// TIA Portal project "OPCUA@SUP_HandsOnProject_V16_Referent" (V16)

(* hardware
DEVICE "S71500/ET200MP-Station_1"  S7-1500 station
   slot 0: "Profilschiene_0"  Rack  6ES7 590-1***0-0AA0
   slot 1: "OPCServer@SUP"  CPU 1518-4 PN/DP  6ES7 518-4AP00-0AB0  V2.8
      slot 3: "CPU-Display_1"  6ES7591-1BA00-0AA0
      slot 32768: "PROFINET-Schnittstelle_1"  X1
      slot 33024: "PROFINET-Schnittstelle_2"  X2
      slot 33280: "PROFINET-Schnittstelle GBIT_3"  X3
      slot 34817: "Virtual CP interface port_1"  Virtual CP interface port  Virtual CP interface port
DEVICE "S71500/ET200MP-Station_2"  S7-1500 station
   slot 0: "Profilschiene_0"  Rack  6ES7 590-1***0-0AA0
   slot 1: "ZOPCClient@SUP"  CPU 1518-4 PN/DP  6ES7 518-4AP00-0AB0  V2.8
      slot 3: "CPU-Display_1"  6ES7591-1BA00-0AA0
      slot 32768: "PROFINET-Schnittstelle_1"  X1
      slot 33024: "PROFINET-Schnittstelle_2"  X2
      slot 33280: "PROFINET-Schnittstelle GBIT_3"  X3
      slot 34817: "Virtual CP interface port_1"  Virtual CP interface port  Virtual CP interface port
*)

// ===== PLC "OPCServer@SUP"  CPU 1518-4 PN/DP =====

VAR_GLOBAL   // PLC tag table "StandardVariablentabelle"
   "ClockByte" AT %MB0 : Byte;
   "Clock10Hz" AT %M0.0 : Bool;
   "Clock5Hz" AT %M0.1 : Bool;
   "Clock2.5Hz" AT %M0.2 : Bool;
   "Clock2Hz" AT %M0.3 : Bool;
   "Clock1.25Hz" AT %M0.4 : Bool;
   "Clock1Hz" AT %M0.5 : Bool;
   "Clock0.625Hz" AT %M0.6 : Bool;
   "Clock0.5Hz" AT %M0.7 : Bool;
   "SystemByte" AT %MB1 : Byte;
   "FirstScan" AT %M1.0 : Bool;
   "DiagStatusUpdate" AT %M1.1 : Bool;
   "AlwaysTRUE" AT %M1.2 : Bool;
   "AlwaysFALSE" AT %M1.3 : Bool;
END_VAR

VAR_GLOBAL   // PLC tag table "AnalogTags"
   "AI0" AT %EW4 : Word;
   "AI1" AT %EW9 : Word;
   "AI2" AT %EW11 : Word;
   "AI3" AT %EW13 : Word;
   "AI4" AT %EW15 : Word;
   "AI5" AT %EW14 : Word;
   "AI6" AT %EW16 : Word;
   "AI7" AT %EW18 : Word;
   "AO0" AT %AW4 : Word;
   "AO1" AT %AW6 : Word;
   "AO2" AT %AW8 : Word;
   "AO3" AT %AW10 : Word;
END_VAR

VAR_GLOBAL   // PLC tag table "CounterTags"
   "Z1" AT %Z1 : Counter;
   "Z2" AT %Z2 : Counter;
   "Z3" AT %Z3 : Counter;
   "Z4" AT %Z4 : Counter;
   "Z5" AT %Z5 : Counter;
   "Z7" AT %Z7 : Counter;
   "Z8" AT %Z8 : Counter;
   "Z9" AT %Z9 : Counter;
   "Z10" AT %Z10 : Counter;
   "ZTest" AT %Z100 : Counter;
   "Z6" AT %Z6 : Counter;
   "Z500" AT %Z500 : Counter;
   "Z1000" AT %Z1000 : Counter;
   "Z1023" AT %Z1023 : Counter;
   "Z1024" AT %Z1024 : Counter;
   "Z2047" AT %Z2047 : Counter;
END_VAR

VAR_GLOBAL   // PLC tag table "DigitalInputTags"
   "DI01" AT %E0.1 : Bool;
   "DI02" AT %E0.2 : Bool;
   "DI03" AT %E0.3 : Bool;
   "DI04" AT %E0.4 : Bool;
   "DI05" AT %E0.5 : Bool;
   "DI06" AT %E0.6 : Bool;
   "DI07" AT %E0.7 : Bool;
   "DI11" AT %E1.1 : Bool;
   "DI12" AT %E1.2 : Bool;
   "DI13" AT %E1.3 : Bool;
   "DI14" AT %E1.4 : Bool;
   "DI15" AT %E1.5 : Bool;
   "DI16" AT %E1.6 : Bool;
   "DI17" AT %E1.7 : Bool;
   "DI20" AT %E2.0 : Bool;
   "DI21" AT %E2.1 : Bool;
   "DI22" AT %E2.2 : Bool;
   "DI23" AT %E2.3 : Bool;
   "DI24" AT %E2.4 : Bool;
   "DI25" AT %E2.5 : Bool;
   "DI26" AT %E2.6 : Bool;
   "DI27" AT %E2.7 : Bool;
   "DI30" AT %E3.0 : Bool;
   "DI31" AT %E3.1 : Bool;
   "DI32" AT %E3.2 : Bool;
   "DI33" AT %E3.3 : Bool;
   "DI34" AT %E3.4 : Bool;
   "DI35" AT %E3.5 : Bool;
   "DI36" AT %E3.6 : Bool;
   "DI37" AT %E3.7 : Bool;
   "DI10" AT %E1.0 : Bool;
   "DI00" AT %E0.0 : Bool;
   "DI1" AT %EB1 : Byte;
   "DI300" AT %EB300 : Byte;
   "DI310W" AT %EW310 : Word;
   "DI320D" AT %ED320 : DWord;
   "DI3300" AT %E330.0 : Bool;
   "DI340L" AT %E340.0 : LWord;
   "DI0" AT %EB0 : Byte;
END_VAR

VAR_GLOBAL   // PLC tag table "DigitalOutputTags"
   "DO01" AT %A0.1 : Bool;
   "DO02" AT %A0.2 : Bool;
   "DO04" AT %A0.4 : Bool;
   "DO05" AT %A0.5 : Bool;
   "DO06" AT %A0.6 : Bool;
   "DO07" AT %A0.7 : Bool;
   "DO10" AT %A1.0 : Bool;
   "DO11" AT %A1.1 : Bool;
   "DO12" AT %A1.2 : Bool;
   "DO13" AT %A1.3 : Bool;
   "DO14" AT %A1.4 : Bool;
   "DO15" AT %A1.5 : Bool;
   "DO16" AT %A1.6 : Bool;
   "DO17" AT %A1.7 : Bool;
   "DO20" AT %A2.0 : Bool;
   "DO21" AT %A2.1 : Bool;
   "DO22" AT %A2.2 : Bool;
   "DO23" AT %A2.3 : Bool;
   "DO24" AT %A2.4 : Bool;
   "DO25" AT %A2.5 : Bool;
   "DO26" AT %A2.6 : Bool;
   "DO27" AT %A2.7 : Bool;
   "DO30" AT %A3.0 : Bool;
   "DO31" AT %A3.1 : Bool;
   "DO32" AT %A3.2 : Bool;
   "DO33" AT %A3.3 : Bool;
   "DO34" AT %A3.4 : Bool;
   "DO35" AT %A3.5 : Bool;
   "DO36" AT %A3.6 : Bool;
   "DO37" AT %A3.7 : Bool;
   "DO300" AT %AB300 : Byte;
   "DO00" AT %A0.0 : Bool;
   "DO03" AT %A0.3 : Bool;
   "DO120" AT %A12.0 : Bool;
   "DO1" AT %AB1 : Byte;
   "DO0" AT %AB0 : Byte;
   "DOW0" AT %AW0 : Word;
   "DOW2" AT %AW2 : Word;
   "DO310W" AT %AW310 : Word;
   "DO320D" AT %AD320 : DWord;
   "DO3300" AT %A330.0 : Bool;
   "DO340L" AT %A340.0 : LWord;
END_VAR

VAR_GLOBAL   // PLC tag table "MerkerTags"
   "M1000" AT %M100.0 : Bool;
   "M1001" AT %M100.1 : Bool;
   "M1002" AT %M100.2 : Bool;
   "M1003" AT %M100.3 : Bool;
   "M1004" AT %M100.4 : Bool;
   "M1005" AT %M100.5 : Bool;
   "M1006" AT %M100.6 : Bool;
   "M1007" AT %M100.7 : Bool;
   "MB110" AT %MB110 : Byte;
   "MW120" AT %MW120 : Word;
   "MD130" AT %MD130 : DWord;
   "CharMb" AT %MB200 : Char;
   "DateMw" AT %MW202 : Date;
   "DintMd" AT %MD204 : DInt;
   "IntMw" AT %MW208 : Int;
   "LdtMl" AT %M210.0 : LDT;
   "LintMl" AT %M218.0 : LInt;
   "LrealMl" AT %M226.0 : LReal;
   "LtimeMl" AT %M234.0 : LTime;
   "LtodMl" AT %M242.0 : LTime_Of_Day;
   "LwordMl" AT %M250.0 : LWord;
   "RealMd" AT %MD258 : Real;
   "S5timeMw" AT %MW262 : S5Time;
   "SintMb" AT %MB264 : SInt;
   "TimeMd" AT %MD266 : Time;
   "TodMd" AT %MD270 : Time_Of_Day;
   "UdintMd" AT %MD274 : UDInt;
   "UintMw" AT %MW278 : UInt;
   "UlintMl" AT %M280.0 : ULInt;
   "UsintMb" AT %MB288 : USInt;
   "Z1MB" AT %MB500 : Byte;
   "Z2MB" AT %MB501 : Byte;
   "ZTestMx" AT %M502.0 : Bool;
   "Z6FP" AT %M502.1 : Bool;
   "Z7FP" AT %M502.2 : Bool;
   "Z8FP" AT %M502.3 : Bool;
   "Z9FP" AT %M502.4 : Bool;
   "Z10FP" AT %M502.5 : Bool;
   "TremMx" AT %M105.0 : Bool;
   "IintMw400" AT %MW400 : Int;
END_VAR

VAR_GLOBAL   // PLC tag table "TimerTags"
   "T1" AT %T1 : Timer;
   "T3" AT %T3 : Timer;
   "T4" AT %T4 : Timer;
   "T5" AT %T5 : Timer;
   "T6" AT %T6 : Timer;
   "T7" AT %T7 : Timer;
   "T9" AT %T9 : Timer;
   "T10" AT %T10 : Timer;
   "T2" AT %T2 : Timer;
   "T8" AT %T8 : Timer;
   "T20" AT %T20 : Timer;
   "T40" AT %T40 : Timer;
   "T60" AT %T60 : Timer;
   "T80" AT %T80 : Timer;
   "T100" AT %T100 : Timer;
   "T200" AT %T200 : Timer;
   "T500" AT %T500 : Timer;
   "T1000" AT %T1000 : Timer;
   "T2000" AT %T2000 : Timer;
   "T99" AT %T99 : Timer;
   "T85" AT %T85 : Timer;
   "T86" AT %T86 : Timer;
   "T2047" AT %T2047 : Timer;
END_VAR

VAR_GLOBAL CONSTANT   // PLC tag table "Tag table from XML_1"
   "OpcUa_Good" : DWord := 16#00000000;   // Everything is as expected.
   "OpcUa_Uncertain" : DWord := 16#40000000;   // Something unexpected occurred but the results still maybe useable.
   "OpcUa_Bad" : DWord := 16#80000000;   // An error occurred.
   "OpcUa_BadUnexpectedError" : DWord := 16#80010000;   // An unexpected error occurred.
   "OpcUa_BadInternalError" : DWord := 16#80020000;   // An internal error occurred as a result of a programming or configuration error.
   "OpcUa_BadOutOfMemory" : DWord := 16#80030000;   // Not enough memory to complete the operation.
   "OpcUa_BadResourceUnavailable" : DWord := 16#80040000;   // An operating system resource is not available.
   "OpcUa_BadCommunicationError" : DWord := 16#80050000;   // A low level communication error occurred.
   "OpcUa_BadEncodingError" : DWord := 16#80060000;   // Encoding halted because of invalid data in the objects being serialized.
   "OpcUa_BadDecodingError" : DWord := 16#80070000;   // Decoding halted because of invalid data in the stream.
   "OpcUa_BadEncodingLimitsExceeded" : DWord := 16#80080000;   // The message encoding/decoding limits imposed by the stack have been exceeded.
   "OpcUa_BadRequestTooLarge" : DWord := 16#80B80000;   // The request message size exceeds limits set by the server.
   "OpcUa_BadResponseTooLarge" : DWord := 16#80B90000;   // The response message size exceeds limits set by the client.
   "OpcUa_BadUnknownResponse" : DWord := 16#80090000;   // An unrecognized response was received from the server.
   "OpcUa_BadTimeout" : DWord := 16#800A0000;   // The operation timed out.
   "OpcUa_BadServiceUnsupported" : DWord := 16#800B0000;   // The server does not support the requested service.
   "OpcUa_BadShutdown" : DWord := 16#800C0000;   // The operation was cancelled because the application is shutting down.
   "OpcUa_BadServerNotConnected" : DWord := 16#800D0000;   // The operation could not complete because the client is not connected to the server.
   "OpcUa_BadServerHalted" : DWord := 16#800E0000;   // The server has stopped and cannot process any requests.
   "OpcUa_BadNothingToDo" : DWord := 16#800F0000;   // There was nothing to do because the client passed a list of operations with no elements.
   "OpcUa_BadTooManyOperations" : DWord := 16#80100000;   // The request could not be processed because it specified too many operations.
   "OpcUa_BadTooManyMonitoredItems" : DWord := 16#80DB0000;   // The request could not be processed because there are too many monitored items in the subscription.
   "OpcUa_BadDataTypeIdUnknown" : DWord := 16#80110000;   // The extension object cannot be (de)serialized because the data type id is not recognized.
   "OpcUa_BadCertificateInvalid" : DWord := 16#80120000;   // The certificate provided as a parameter is not valid.
   "OpcUa_BadSecurityChecksFailed" : DWord := 16#80130000;   // An error occurred verifying security.
   "OpcUa_BadCertificateTimeInvalid" : DWord := 16#80140000;   // The certificate has expired or is not yet valid.
   "OpcUa_BadCertificateIssuerTimeInvalid" : DWord := 16#80150000;   // An issuer certificate has expired or is not yet valid.
   "OpcUa_BadCertificateHostNameInvalid" : DWord := 16#80160000;   // The HostName used to connect to a server does not match a HostName in the certificate.
   "OpcUa_BadCertificateUriInvalid" : DWord := 16#80170000;   // The URI specified in the ApplicationDescription does not match the URI in the certificate.
   "OpcUa_BadCertificateUseNotAllowed" : DWord := 16#80180000;   // The certificate may not be used for the requested operation.
   "OpcUa_BadCertificateIssuerUseNotAllowed" : DWord := 16#80190000;   // The issuer certificate may not be used for the requested operation.
   "OpcUa_BadCertificateUntrusted" : DWord := 16#801A0000;   // The certificate is not trusted.
   "OpcUa_BadCertificateRevocationUnknown" : DWord := 16#801B0000;   // It was not possible to determine if the certificate has been revoked.
   "OpcUa_BadCertificateIssuerRevocationUnknown" : DWord := 16#801C0000;   // It was not possible to determine if the issuer certificate has been revoked.
   "OpcUa_BadCertificateRevoked" : DWord := 16#801D0000;   // The certificate has been revoked.
   "OpcUa_BadCertificateIssuerRevoked" : DWord := 16#801E0000;   // The issuer certificate has been revoked.
   "OpcUa_BadCertificateChainIncomplete" : DWord := 16#810D0000;   // The certificate chain is incomplete.
   "OpcUa_BadUserAccessDenied" : DWord := 16#801F0000;   // User does not have permission to perform the requested operation.
   "OpcUa_BadIdentityTokenInvalid" : DWord := 16#80200000;   // The user identity token is not valid.
   "OpcUa_BadIdentityTokenRejected" : DWord := 16#80210000;   // The user identity token is valid but the server has rejected it.
   "OpcUa_BadSecureChannelIdInvalid" : DWord := 16#80220000;   // The specified secure channel is no longer valid.
   "OpcUa_BadInvalidTimestamp" : DWord := 16#80230000;   // The timestamp is outside the range allowed by the server.
   "OpcUa_BadNonceInvalid" : DWord := 16#80240000;   // The nonce does appear to be not a random value or it is not the correct length.
   "OpcUa_BadSessionIdInvalid" : DWord := 16#80250000;   // The session id is not valid.
   "OpcUa_BadSessionClosed" : DWord := 16#80260000;   // The session was closed by the client.
   "OpcUa_BadSessionNotActivated" : DWord := 16#80270000;   // The session cannot be used because ActivateSession has not been called.
   "OpcUa_BadSubscriptionIdInvalid" : DWord := 16#80280000;   // The subscription id is not valid.
   "OpcUa_BadRequestHeaderInvalid" : DWord := 16#802A0000;   // The header for the request is missing or invalid.
   "OpcUa_BadTimestampsToReturnInvalid" : DWord := 16#802B0000;   // The timestamps to return parameter is invalid.
   "OpcUa_BadRequestCancelledByClient" : DWord := 16#802C0000;   // The request was cancelled by the client.
   "OpcUa_BadTooManyArguments" : DWord := 16#80E50000;   // Too many arguments were provided.
   "OpcUa_BadLicenseExpired" : DWord := 16#810E0000;   // The server requires a license to operate in general or to perform a service or operation, but existing license is expired.
   "OpcUa_BadLicenseLimitsExceeded" : DWord := 16#810F0000;   // The server has limits on number of allowed operations / objects, based on installed licenses, and these limits where exceeded.
   "OpcUa_BadLicenseNotAvailable" : DWord := 16#81100000;   // The server does not have a license which is required to operate in general or to perform a service or operation.
   "OpcUa_GoodSubscriptionTransferred" : DWord := 16#002D0000;   // The subscription was transferred to another session.
   "OpcUa_GoodCompletesAsynchronously" : DWord := 16#002E0000;   // The processing will complete asynchronously.
   "OpcUa_GoodOverload" : DWord := 16#002F0000;   // Sampling has slowed down due to resource limitations.
   "OpcUa_GoodClamped" : DWord := 16#00300000;   // The value written was accepted but was clamped.
   "OpcUa_BadNoCommunication" : DWord := 16#80310000;   // Communication with the data source is defined, but not established, and there is no last known value available.
   "OpcUa_BadWaitingForInitialData" : DWord := 16#80320000;   // Waiting for the server to obtain values from the underlying data source.
   "OpcUa_BadNodeIdInvalid" : DWord := 16#80330000;   // The syntax of the node id is not valid.
   "OpcUa_BadNodeIdUnknown" : DWord := 16#80340000;   // The node id refers to a node that does not exist in the server address space.
   "OpcUa_BadAttributeIdInvalid" : DWord := 16#80350000;   // The attribute is not supported for the specified Node.
   "OpcUa_BadIndexRangeInvalid" : DWord := 16#80360000;   // The syntax of the index range parameter is invalid.
   "OpcUa_BadIndexRangeNoData" : DWord := 16#80370000;   // No data exists within the range of indexes specified.
   "OpcUa_BadDataEncodingInvalid" : DWord := 16#80380000;   // The data encoding is invalid.
   "OpcUa_BadDataEncodingUnsupported" : DWord := 16#80390000;   // The server does not support the requested data encoding for the node.
   "OpcUa_BadNotReadable" : DWord := 16#803A0000;   // The access level does not allow reading or subscribing to the Node.
   "OpcUa_BadNotWritable" : DWord := 16#803B0000;   // The access level does not allow writing to the Node.
   "OpcUa_BadOutOfRange" : DWord := 16#803C0000;   // The value was out of range.
   "OpcUa_BadNotSupported" : DWord := 16#803D0000;   // The requested operation is not supported.
   "OpcUa_BadNotFound" : DWord := 16#803E0000;   // A requested item was not found or a search operation ended without success.
   "OpcUa_BadObjectDeleted" : DWord := 16#803F0000;   // The object cannot be used because it has been deleted.
   "OpcUa_BadNotImplemented" : DWord := 16#80400000;   // Requested operation is not implemented.
   "OpcUa_BadMonitoringModeInvalid" : DWord := 16#80410000;   // The monitoring mode is invalid.
   "OpcUa_BadMonitoredItemIdInvalid" : DWord := 16#80420000;   // The monitoring item id does not refer to a valid monitored item.
   "OpcUa_BadMonitoredItemFilterInvalid" : DWord := 16#80430000;   // The monitored item filter parameter is not valid.
   "OpcUa_BadMonitoredItemFilterUnsupported" : DWord := 16#80440000;   // The server does not support the requested monitored item filter.
   "OpcUa_BadFilterNotAllowed" : DWord := 16#80450000;   // A monitoring filter cannot be used in combination with the attribute specified.
   "OpcUa_BadStructureMissing" : DWord := 16#80460000;   // A mandatory structured parameter was missing or null.
   "OpcUa_BadEventFilterInvalid" : DWord := 16#80470000;   // The event filter is not valid.
   "OpcUa_BadContentFilterInvalid" : DWord := 16#80480000;   // The content filter is not valid.
   "OpcUa_BadFilterOperatorInvalid" : DWord := 16#80C10000;   // An unregognized operator was provided in a filter.
   "OpcUa_BadFilterOperatorUnsupported" : DWord := 16#80C20000;   // A valid operator was provided, but the server does not provide support for this filter operator.
   "OpcUa_BadFilterOperandCountMismatch" : DWord := 16#80C30000;   // The number of operands provided for the filter operator was less then expected for the operand provided.
   "OpcUa_BadFilterOperandInvalid" : DWord := 16#80490000;   // The operand used in a content filter is not valid.
   "OpcUa_BadFilterElementInvalid" : DWord := 16#80C40000;   // The referenced element is not a valid element in the content filter.
   "OpcUa_BadFilterLiteralInvalid" : DWord := 16#80C50000;   // The referenced literal is not a valid value.
   "OpcUa_BadContinuationPointInvalid" : DWord := 16#804A0000;   // The continuation point provide is longer valid.
   "OpcUa_BadNoContinuationPoints" : DWord := 16#804B0000;   // The operation could not be processed because all continuation points have been allocated.
   "OpcUa_BadReferenceTypeIdInvalid" : DWord := 16#804C0000;   // The operation could not be processed because all continuation points have been allocated.
   "OpcUa_BadBrowseDirectionInvalid" : DWord := 16#804D0000;   // The browse direction is not valid.
   "OpcUa_BadNodeNotInView" : DWord := 16#804E0000;   // The node is not part of the view.
   "OpcUa_BadNumericOverflow" : DWord := 16#81120000;   // The number was not accepted because of a numeric overflow.
   "OpcUa_BadServerUriInvalid" : DWord := 16#804F0000;   // The ServerUri is not a valid URI.
   "OpcUa_BadServerNameMissing" : DWord := 16#80500000;   // No ServerName was specified.
   "OpcUa_BadDiscoveryUrlMissing" : DWord := 16#80510000;   // No DiscoveryUrl was specified.
   "OpcUa_BadSempahoreFileMissing" : DWord := 16#80520000;   // The semaphore file specified by the client is not valid.
   "OpcUa_BadRequestTypeInvalid" : DWord := 16#80530000;   // The security token request type is not valid.
   "OpcUa_BadSecurityModeRejected" : DWord := 16#80540000;   // The security mode does not meet the requirements set by the server.
   "OpcUa_BadSecurityPolicyRejected" : DWord := 16#80550000;   // The security policy does not meet the requirements set by the server.
   "OpcUa_BadTooManySessions" : DWord := 16#80560000;   // The server has reached its maximum number of sessions.
   "OpcUa_BadUserSignatureInvalid" : DWord := 16#80570000;   // The user token signature is missing or invalid.
   "OpcUa_BadApplicationSignatureInvalid" : DWord := 16#80580000;   // The signature generated with the client certificate is missing or invalid.
   "OpcUa_BadNoValidCertificates" : DWord := 16#80590000;   // The client did not provide at least one software certificate that is valid and meets the profile requirements for the server.
   "OpcUa_BadIdentityChangeNotSupported" : DWord := 16#80C60000;   // The server does not support changing the user identity assigned to the session.
   "OpcUa_BadRequestCancelledByRequest" : DWord := 16#805A0000;   // The request was cancelled by the client with the Cancel service.
   "OpcUa_BadParentNodeIdInvalid" : DWord := 16#805B0000;   // The parent node id does not to refer to a valid node.
   "OpcUa_BadReferenceNotAllowed" : DWord := 16#805C0000;   // The reference could not be created because it violates constraints imposed by the data model.
   "OpcUa_BadNodeIdRejected" : DWord := 16#805D0000;   // The requested node id was reject because it was either invalid or server does not allow node ids to be specified by the client.
   "OpcUa_BadNodeIdExists" : DWord := 16#805E0000;   // The requested node id is already used by another node.
   "OpcUa_BadNodeClassInvalid" : DWord := 16#805F0000;   // The node class is not valid.
   "OpcUa_BadBrowseNameInvalid" : DWord := 16#80600000;   // The browse name is invalid.
   "OpcUa_BadBrowseNameDuplicated" : DWord := 16#80610000;   // The browse name is not unique among nodes that share the same relationship with the parent.
   "OpcUa_BadNodeAttributesInvalid" : DWord := 16#80620000;   // The node attributes are not valid for the node class.
   "OpcUa_BadTypeDefinitionInvalid" : DWord := 16#80630000;   // The type definition node id does not reference an appropriate type node.
   "OpcUa_BadSourceNodeIdInvalid" : DWord := 16#80640000;   // The source node id does not reference a valid node.
   "OpcUa_BadTargetNodeIdInvalid" : DWord := 16#80650000;   // The target node id does not reference a valid node.
   "OpcUa_BadDuplicateReferenceNotAllowed" : DWord := 16#80660000;   // The reference type between the nodes is already defined.
   "OpcUa_BadInvalidSelfReference" : DWord := 16#80670000;   // The server does not allow this type of self reference on this node.
   "OpcUa_BadReferenceLocalOnly" : DWord := 16#80680000;   // The reference type is not valid for a reference to a remote server.
   "OpcUa_BadNoDeleteRights" : DWord := 16#80690000;   // The server will not allow the node to be deleted.
   "OpcUa_UncertainReferenceNotDeleted" : DWord := 16#40BC0000;   // The server was not able to delete all target references.
   "OpcUa_BadServerIndexInvalid" : DWord := 16#806A0000;   // The server index is not valid.
   "OpcUa_BadViewIdUnknown" : DWord := 16#806B0000;   // The view id does not refer to a valid view node.
   "OpcUa_BadViewTimestampInvalid" : DWord := 16#80C90000;   // The view timestamp is not available or not supported.
   "OpcUa_BadViewParameterMismatch" : DWord := 16#80CA0000;   // The view parameters are not consistent with each other.
   "OpcUa_BadViewVersionInvalid" : DWord := 16#80CB0000;   // The view version is not available or not supported.
   "OpcUa_UncertainNotAllNodesAvailable" : DWord := 16#40C00000;   // The list of references may not be complete because the underlying system is not available.
   "OpcUa_GoodResultsMayBeIncomplete" : DWord := 16#00BA0000;   // The server should have followed a reference to a node in a remote server but did not. The result set may be incomplete.
   "OpcUa_BadNotTypeDefinition" : DWord := 16#80C80000;   // The provided Nodeid was not a type definition nodeid.
   "OpcUa_UncertainReferenceOutOfServer" : DWord := 16#406C0000;   // One of the references to follow in the relative path references to a node in the address space in another server.
   "OpcUa_BadTooManyMatches" : DWord := 16#806D0000;   // The requested operation has too many matches to return.
   "OpcUa_BadQueryTooComplex" : DWord := 16#806E0000;   // The requested operation requires too many resources in the server.
   "OpcUa_BadNoMatch" : DWord := 16#806F0000;   // The requested operation has no match to return.
   "OpcUa_BadMaxAgeInvalid" : DWord := 16#80700000;   // The max age parameter is invalid.
   "OpcUa_BadSecurityModeInsufficient" : DWord := 16#80E60000;   // The operation is not permitted over the current secure channel.
   "OpcUa_BadHistoryOperationInvalid" : DWord := 16#80710000;   // The history details parameter is not valid.
   "OpcUa_BadHistoryOperationUnsupported" : DWord := 16#80720000;   // The server does not support the requested operation.
   "OpcUa_BadInvalidTimestampArgument" : DWord := 16#80BD0000;   // The defined timestamp to return was invalid.
   "OpcUa_BadWriteNotSupported" : DWord := 16#80730000;   // The server does not support writing the combination of value, status and timestamps provided.
   "OpcUa_BadTypeMismatch" : DWord := 16#80740000;   // The value supplied for the attribute is not of the same type as the attributes value.
   "OpcUa_BadMethodInvalid" : DWord := 16#80750000;   // The method id does not refer to a method for the specified object.
   "OpcUa_BadArgumentsMissing" : DWord := 16#80760000;   // The client did not specify all of the input arguments for the method.
   "OpcUa_BadNotExecutable" : DWord := 16#81110000;   // The executable attribute does not allow the execution of the method.
   "OpcUa_BadTooManySubscriptions" : DWord := 16#80770000;   // The server has reached its maximum number of subscriptions.
   "OpcUa_BadTooManyPublishRequests" : DWord := 16#80780000;   // The server has reached the maximum number of queued publish requests.
   "OpcUa_BadNoSubscription" : DWord := 16#80790000;   // There is no subscription available for this session.
   "OpcUa_BadSequenceNumberUnknown" : DWord := 16#807A0000;   // The sequence number is unknown to the server.
   "OpcUa_BadMessageNotAvailable" : DWord := 16#807B0000;   // The requested notification message is no longer available.
   "OpcUa_BadInsufficientClientProfile" : DWord := 16#807C0000;   // The client of the current session does not support one or more Profiles that are necessary for the subscription.
   "OpcUa_BadStateNotActive" : DWord := 16#80BF0000;   // The sub-state machine is not currently active.
   "OpcUa_BadTcpServerTooBusy" : DWord := 16#807D0000;   // The server cannot process the request because it is too busy.
   "OpcUa_BadTcpMessageTypeInvalid" : DWord := 16#807E0000;   // The type of the message specified in the header invalid.
   "OpcUa_BadTcpSecureChannelUnknown" : DWord := 16#807F0000;   // The SecureChannelId and/or TokenId are not currently in use.
   "OpcUa_BadTcpMessageTooLarge" : DWord := 16#80800000;   // The size of the message specified in the header is too large.
   "OpcUa_BadTcpNotEnoughResources" : DWord := 16#80810000;   // There are not enough resources to process the request.
   "OpcUa_BadTcpInternalError" : DWord := 16#80820000;   // An internal error occurred.
   "OpcUa_BadTcpEndpointUrlInvalid" : DWord := 16#80830000;   // The server does not recognize the QueryString specified.
   "OpcUa_BadRequestInterrupted" : DWord := 16#80840000;   // The request could not be sent because of a network interruption.
   "OpcUa_BadRequestTimeout" : DWord := 16#80850000;   // Timeout occurred while processing the request.
   "OpcUa_BadSecureChannelClosed" : DWord := 16#80860000;   // The secure channel has been closed.
   "OpcUa_BadSecureChannelTokenUnknown" : DWord := 16#80870000;   // The token has expired or is not recognized.
   "OpcUa_BadSequenceNumberInvalid" : DWord := 16#80880000;   // The sequence number is not valid.
   "OpcUa_BadProtocolVersionUnsupported" : DWord := 16#80BE0000;   // The applications do not have compatible protocol versions.
   "OpcUa_BadConfigurationError" : DWord := 16#80890000;   // There is a problem with the configuration that affects the usefulness of the value.
   "OpcUa_BadNotConnected" : DWord := 16#808A0000;   // The variable should receive its value from another variable, but has never been configured to do so.
   "OpcUa_BadDeviceFailure" : DWord := 16#808B0000;   // There has been a failure in the device/data source that generates the value that has affected the value.
   "OpcUa_BadSensorFailure" : DWord := 16#808C0000;   // There has been a failure in the sensor from which the value is derived by the device/data source.
   "OpcUa_BadOutOfService" : DWord := 16#808D0000;   // The source of the data is not operational.
   "OpcUa_BadDeadbandFilterInvalid" : DWord := 16#808E0000;   // The deadband filter is not valid.
   "OpcUa_UncertainNoCommunicationLastUsableValue" : DWord := 16#408F0000;   // Communication to the data source has failed. The variable value is the last value that had a good quality.
   "OpcUa_UncertainLastUsableValue" : DWord := 16#40900000;   // Whatever was updating this value has stopped doing so.
   "OpcUa_UncertainSubstituteValue" : DWord := 16#40910000;   // The value is an operational value that was manually overwritten.
   "OpcUa_UncertainInitialValue" : DWord := 16#40920000;   // The value is an initial value for a variable that normally receives its value from another variable.
   "OpcUa_UncertainSensorNotAccurate" : DWord := 16#40930000;   // The value is at one of the sensor limits.
   "OpcUa_UncertainEngineeringUnitsExceeded" : DWord := 16#40940000;   // The value is outside of the range of values defined for this parameter.
   "OpcUa_UncertainSubNormal" : DWord := 16#40950000;   // The value is derived from multiple sources and has less than the required number of Good sources.
   "OpcUa_GoodLocalOverride" : DWord := 16#00960000;   // The value has been overridden.
   "OpcUa_BadRefreshInProgress" : DWord := 16#80970000;   // This Condition refresh failed, a Condition refresh operation is already in progress.
   "OpcUa_BadConditionAlreadyDisabled" : DWord := 16#80980000;   // This condition has already been disabled.
   "OpcUa_BadConditionAlreadyEnabled" : DWord := 16#80CC0000;   // This condition has already been enabled.
   "OpcUa_BadConditionDisabled" : DWord := 16#80990000;   // Property not available, this condition is disabled.
   "OpcUa_BadEventIdUnknown" : DWord := 16#809A0000;   // The specified event id is not recognized.
   "OpcUa_BadEventNotAcknowledgeable" : DWord := 16#80BB0000;   // The event cannot be acknowledged.
   "OpcUa_BadDialogNotActive" : DWord := 16#80CD0000;   // The dialog condition is not active.
   "OpcUa_BadDialogResponseInvalid" : DWord := 16#80CE0000;   // The response is not valid for the dialog.
   "OpcUa_BadConditionBranchAlreadyAcked" : DWord := 16#80CF0000;   // The condition branch has already been acknowledged.
   "OpcUa_BadConditionBranchAlreadyConfirmed" : DWord := 16#80D00000;   // The condition branch has already been confirmed.
   "OpcUa_BadConditionAlreadyShelved" : DWord := 16#80D10000;   // The condition has already been shelved.
   "OpcUa_BadConditionNotShelved" : DWord := 16#80D20000;   // The condition is not currently shelved.
   "OpcUa_BadShelvingTimeOutOfRange" : DWord := 16#80D30000;   // The shelving time not within an acceptable range.
   "OpcUa_BadNoData" : DWord := 16#809B0000;   // No data exists for the requested time range or event filter.
   "OpcUa_BadBoundNotFound" : DWord := 16#80D70000;   // No data found to provide upper or lower bound value.
   "OpcUa_BadBoundNotSupported" : DWord := 16#80D80000;   // The server cannot retrieve a bound for the variable.
   "OpcUa_BadDataLost" : DWord := 16#809D0000;   // Data is missing due to collection started/stopped/lost.
   "OpcUa_BadDataUnavailable" : DWord := 16#809E0000;   // Expected data is unavailable for the requested time range due to an un-mounted volume, an off-line archive or tape, or similar reason for temporary unavailability.
   "OpcUa_BadEntryExists" : DWord := 16#809F0000;   // The data or event was not successfully inserted because a matching entry exists.
   "OpcUa_BadNoEntryExists" : DWord := 16#80A00000;   // The data or event was not successfully updated because no matching entry exists.
   "OpcUa_BadTimestampNotSupported" : DWord := 16#80A10000;   // The client requested history using a timestamp format the server does not support (i.e requested ServerTimestamp when server only supports SourceTimestamp).
   "OpcUa_GoodEntryInserted" : DWord := 16#00A20000;   // The data or event was successfully inserted into the historical database.
   "OpcUa_GoodEntryReplaced" : DWord := 16#00A30000;   // The data or event field was successfully replaced in the historical database.
   "OpcUa_UncertainDataSubNormal" : DWord := 16#40A40000;   // The value is derived from multiple values and has less than the required number of Good values.
   "OpcUa_GoodNoData" : DWord := 16#00A50000;   // No data exists for the requested time range or event filter.
   "OpcUa_GoodMoreData" : DWord := 16#00A60000;   // The data or event field was successfully replaced in the historical database.
   "OpcUa_BadAggregateListMismatch" : DWord := 16#80D40000;   // The requested number of Aggregates does not match the requested number of NodeIds.
   "OpcUa_BadAggregateNotSupported" : DWord := 16#80D50000;   // The requested Aggregate is not support by the server.
   "OpcUa_BadAggregateInvalidInputs" : DWord := 16#80D60000;   // The aggregate value could not be derived due to invalid data inputs.
   "OpcUa_BadAggregateConfigurationRejected" : DWord := 16#80DA0000;   // The aggregate configuration is not valid for specified node.
   "OpcUa_GoodDataIgnored" : DWord := 16#00D90000;   // The request pecifies fields which are not valid for the EventType or cannot be saved by the historian.
   "OpcUa_BadRequestNotAllowed" : DWord := 16#80E40000;   // The request was rejected by the server because it did not meet the criteria set by the server.
   "OpcUa_BadRequestNotComplete" : DWord := 16#81130000;   // The request has not been processed by the server yet.
   "OpcUa_GoodEdited" : DWord := 16#00DC0000;   // The value does not come from the real source and has been edited by the server.
   "OpcUa_GoodPostActionFailed" : DWord := 16#00DD0000;   // There was an error in execution of these post-actions.
   "OpcUa_UncertainDominantValueChanged" : DWord := 16#40DE0000;   // The related EngineeringUnit has been changed but the Variable Value is still provided based on the previous unit.
   "OpcUa_GoodDependentValueChanged" : DWord := 16#00E00000;   // A dependent value has been changed but the change has not been applied to the device.
   "OpcUa_BadDominantValueChanged" : DWord := 16#80E10000;   // The related EngineeringUnit has been changed but this change has not been applied to the device. The Variable Value is still dependent on the previous unit but its status is currently Bad.
   "OpcUa_UncertainDependentValueChanged" : DWord := 16#40E20000;   // A dependent value has been changed but the change has not been applied to the device. The quality of the dominant variable is uncertain.
   "OpcUa_BadDependentValueChanged" : DWord := 16#80E30000;   // A dependent value has been changed but the change has not been applied to the device. The quality of the dominant variable is Bad.
   "OpcUa_GoodCommunicationEvent" : DWord := 16#00A70000;   // The communication layer has raised an event.
   "OpcUa_GoodShutdownEvent" : DWord := 16#00A80000;   // The system is shutting down.
   "OpcUa_GoodCallAgain" : DWord := 16#00A90000;   // The operation is not finished and needs to be called again.
   "OpcUa_GoodNonCriticalTimeout" : DWord := 16#00AA0000;   // A non-critical timeout occurred.
   "OpcUa_BadInvalidArgument" : DWord := 16#80AB0000;   // One or more arguments are invalid.
   "OpcUa_BadConnectionRejected" : DWord := 16#80AC0000;   // Could not establish a network connection to remote server.
   "OpcUa_BadDisconnect" : DWord := 16#80AD0000;   // The server has disconnected from the client.
   "OpcUa_BadConnectionClosed" : DWord := 16#80AE0000;   // The network connection has been closed.
   "OpcUa_BadInvalidState" : DWord := 16#80AF0000;   // The operation cannot be completed because the object is closed, uninitialized or in some other invalid state.
   "OpcUa_BadEndOfStream" : DWord := 16#80B00000;   // Cannot move beyond end of the stream.
   "OpcUa_BadNoDataAvailable" : DWord := 16#80B10000;   // No data is currently available for reading from a non-blocking stream.
   "OpcUa_BadWaitingForResponse" : DWord := 16#80B20000;   // The asynchronous operation is waiting for a response.
   "OpcUa_BadOperationAbandoned" : DWord := 16#80B30000;   // The asynchronous operation was abandoned by the caller.
   "OpcUa_BadExpectedStreamToBlock" : DWord := 16#80B40000;   // The stream did not return all data requested (possibly because it is a non-blocking stream).
   "OpcUa_BadWouldBlock" : DWord := 16#80B50000;   // Non blocking behaviour is required and the operation would block.
   "OpcUa_BadSyntaxError" : DWord := 16#80B60000;   // A value had an invalid syntax.
   "OpcUa_BadMaxConnectionsReached" : DWord := 16#80B70000;   // The operation could not be finished because all available connections are in use.
END_VAR

TYPE "typeToolParameter"
   STRUCT
      length : Int;
      width : Int;
      weight : Int;
      toolID : Int;
   END_STRUCT;
END_TYPE

// folder: 03_Basics/Process

DATA_BLOCK "InstHMISimulation"   // DB7
{ S7_Optimized_Access := 'TRUE' }
VERSION : 0.1
// stored: InstanceOfName HMISimulation
"HMISimulation"
BEGIN
END_DATA_BLOCK

DATA_BLOCK "InstMachineSimulation"   // DB8
{ S7_Optimized_Access := 'TRUE' }
VERSION : 0.1
// stored: InstanceOfName MachineSimulation
"MachineSimulation"
BEGIN
END_DATA_BLOCK

// folder: 03_Basics/datablocks

DATA_BLOCK "MachineData"   // DB1
{ S7_Optimized_Access := 'TRUE' }
VERSION : 0.1
   VAR
      Manufacturer : WString := WSTRING#'Siemens';
      Operator : WString := WSTRING#'Otello';
      SerialNumber : DWord := 16#12345678;
      "Type" : DInt := 14;
      Fun : Bool := true;
   END_VAR
BEGIN
END_DATA_BLOCK

DATA_BLOCK "MachineParameter"   // DB2
{ S7_Optimized_Access := 'TRUE' }
VERSION : 0.1
   VAR
      Speed : LReal;
      Parts : DInt;
      Frequency : Real;
   END_VAR
BEGIN
END_DATA_BLOCK

DATA_BLOCK "MachineStatus"   // DB3
{ S7_Optimized_Access := 'TRUE' }
VERSION : 0.1
   VAR
      StatusRunning : Bool;
      StatusLoad : Int;
      StatusFlow : Real;
   END_VAR
BEGIN
END_DATA_BLOCK

DATA_BLOCK "MachineControl"   // DB4
{ S7_Optimized_Access := 'TRUE' }
VERSION : 0.1
   VAR
      Run : Bool;
      State : Int;
      hmi : Bool := true;
   END_VAR
BEGIN
END_DATA_BLOCK

DATA_BLOCK "HMI"   // DB5
{ S7_Optimized_Access := 'TRUE' }
VERSION : 0.1
   VAR
      TempHigh : Real;
      TempLow : Real;
      Alarm_Activ : Bool;
      Alarm_Message : WString;
   END_VAR
BEGIN
END_DATA_BLOCK

DATA_BLOCK "ToolParameter"   // DB6
{ S7_Optimized_Access := 'TRUE' }
VERSION : 0.1
   VAR
      Param : "typeToolParameter";
   END_VAR
BEGIN
END_DATA_BLOCK

// folder: 05_Methoden

DATA_BLOCK "InstSetParameter"   // DB9
{ S7_Optimized_Access := 'TRUE' }
VERSION : 0.1
// stored: InstanceOfName SetParameter
"SetParameter"
BEGIN
END_DATA_BLOCK

// folder: (top level)

ORGANIZATION_BLOCK "Main"   // OB1, FBD, ProgramCycle
TITLE = "Main Program Sweep (Cycle)"
{ S7_Optimized_Access := 'TRUE' }
VERSION : 0.1
   VAR_INPUT
      Initial_Call : Bool;   // Initial call of this OB
      Remanence : Bool;   // =True, if remanent data are available
   END_VAR
BEGIN

REGION Network 2
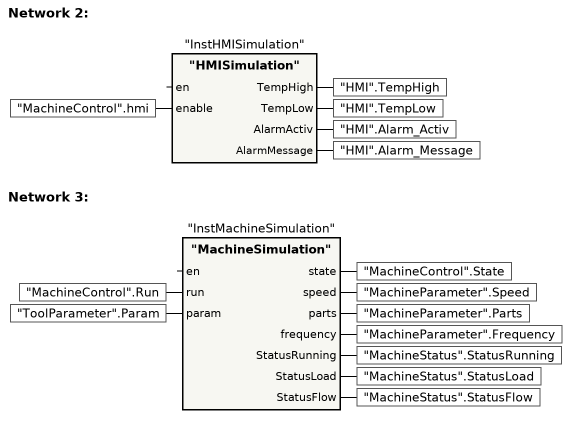
   "InstHMISimulation"(enable := "MachineControl".hmi,   // "HMISimulation"
                       TempHigh => "HMI".TempHigh,
                       TempLow => "HMI".TempLow,
                       AlarmActiv => "HMI".Alarm_Activ,
                       AlarmMessage => "HMI".Alarm_Message);
END_REGION

REGION Network 3
   "InstMachineSimulation"(run := "MachineControl".Run,   // "MachineSimulation"
                           param := "ToolParameter".Param,
                           state => "MachineControl".State,
                           speed => "MachineParameter".Speed,
                           parts => "MachineParameter".Parts,
                           frequency => "MachineParameter".Frequency,
                           StatusRunning => "MachineStatus".StatusRunning,
                           StatusLoad => "MachineStatus".StatusLoad,
                           StatusFlow => "MachineStatus".StatusFlow);
END_REGION
END_ORGANIZATION_BLOCK

ORGANIZATION_BLOCK "Startup"   // OB100, SCL, Startup
TITLE = "Complete Restart"
{ S7_Optimized_Access := 'TRUE' }
VERSION : 0.1
   VAR_INPUT
      LostRetentive : Bool;   // True if retentive data are lost
      LostRTC : Bool;   // True if date and time are lost
   END_VAR
   VAR_TEMP
      temptoolparam : "typeToolParameter";
   END_VAR
BEGIN
   "ToolParameter".Param := #temptoolparam; //Init default
END_ORGANIZATION_BLOCK

// folder: 03_Basics/Process

FUNCTION_BLOCK "MachineSimulation"   // FB1, FBD
{ S7_Optimized_Access := 'TRUE' }
VERSION : 0.1
   VAR_INPUT
      run : Bool;
   END_VAR
   VAR_OUTPUT
      state : Int;
      speed : LReal;
      parts : DInt;
      frequency : Real;
      StatusRunning : Bool;
      StatusLoad : Int;
      StatusFlow : Real;
   END_VAR
   VAR_IN_OUT
      param : "typeToolParameter";
   END_VAR
   VAR
      statstate : Int;
      statspeed : LReal;
      statparts : DInt;
      statfrequency : Real;
      statStatusRunning : Bool;
      statStatusLoad : Int;
      statStatusFlow : Real;
      statArray : Array[0..1] of Bool;
      statlen : Int;
      statwidth : Int;
      statweight : Int;
      statinstTimer : TON_TIME;
      statEmptyArray : Array[0..1] of Bool;
   END_VAR
   VAR CONSTANT
      TIMER_TIMER : Time := t#1s;
   END_VAR
BEGIN

REGION Network 2 (SCL)
   IF #run
   THEN
       #statinstTimer(IN:=#run,
                      PT:=#TIMER_TIMER);
       #statStatusRunning := TRUE;

       IF #statinstTimer.Q
       THEN
           RESET_TIMER(#statinstTimer);

           #statstate := 20;
           #statspeed += 1;
           #statparts += 1;
           #statfrequency += 1;
           #statStatusLoad += 1;
           #statStatusFlow += 1;

           ;

       END_IF;

       #statArray[#param.toolID] := TRUE;

       ;
   ELSE
       #statstate := 10;
       #statspeed := 123.456;
       #statparts := 200;
       #statfrequency := 987.654;
       #statStatusLoad := 20;
       #statStatusFlow := 23.532;
       #statStatusRunning := FALSE;

       #statArray := #statEmptyArray;

       ;
   END_IF;




   #state := #statstate;
   #speed := #statspeed;
   #parts := #statparts;
   #frequency := #statfrequency;
   #StatusRunning := #statStatusRunning;
   #StatusLoad := #statStatusLoad;
   #StatusFlow := #statStatusFlow;
END_REGION
END_FUNCTION_BLOCK

FUNCTION_BLOCK "HMISimulation"   // FB2, FBD
{ S7_Optimized_Access := 'TRUE' }
VERSION : 0.1
   VAR_INPUT
      enable : Bool;
   END_VAR
   VAR_OUTPUT
      TempHigh : Real;
      TempLow : Real;
      AlarmActiv : Bool;
      AlarmMessage : WString;
   END_VAR
   VAR
      statTempTimer : TON_TIME;
      statHigh : Real;
      statLow : Real;
      statAlarm : Bool;
      statAlarmMessage : WString;
   END_VAR
   VAR CONSTANT
      TIME_TIMER : Time := t#3s;
      EMPTY : WString;
      TOO_HIGH : WString := WSTRING#'Temperature too high! attention!';
      TOO_LOW : WString := WSTRING#'Tempearture too low. Attention!';
   END_VAR
BEGIN

REGION Network 2 (SCL)
   IF #enable
   THEN

       #statTempTimer(IN := #enable,
                      PT := #TIME_TIMER
       );

       IF #statTempTimer.Q
       THEN
           #statHigh += 10;
           #statLow -= 5;
           RESET_TIMER(#statTempTimer);

           ;
       END_IF;

       IF #statHigh > 200
       THEN
           #statAlarmMessage := #TOO_HIGH;
           #statAlarm := TRUE;
       ELSIF #statLow < -100
       THEN
           #statAlarmMessage := #TOO_LOW;
           #statAlarm := TRUE;
       END_IF;

       IF #statHigh > 10000 THEN
           #statHigh := 0;
       END_IF;
       IF #statLow < -10000
       THEN
           #statLow := 0;
       END_IF;

   ELSE
       #statHigh := 100;
       #statLow := 0;
       #statAlarm := false;
       #statAlarmMessage := #EMPTY;

   END_IF;

   #TempHigh := #statHigh;
   #TempLow := #statLow;
   #AlarmActiv := #statAlarm;
   #AlarmMessage := #statAlarmMessage;
END_REGION
END_FUNCTION_BLOCK

// folder: 05_Methoden

FUNCTION_BLOCK "SetParameter"   // FB3, FBD
{ S7_Optimized_Access := 'TRUE' }
VERSION : 0.1
   VAR_INPUT
      disabled : Bool;
   END_VAR
   VAR_IN_OUT
      ToolParameter : "typeToolParameter";
   END_VAR
   VAR
      OPC_UA_ServerMethodPre_Instance : OPC_UA_ServerMethodPre;
      OPC_UA_ServerMethodPost_Instance : OPC_UA_ServerMethodPost;
      UAMethod_InParameters : Struct
         ToolParameter : "typeToolParameter";
      END_STRUCT;
      UAMethod_OutParameters : Struct
         Valid : Bool;
      END_STRUCT;
   END_VAR
   VAR_TEMP
      tempMethCalled : Bool;
      tempMethFinished : Bool;
      tempMethResult : DWord;
   END_VAR
   VAR CONSTANT
      MAX_TOOL_ID : Int := 1;
      NULL_ID : Int := 0;
      FALSE : Bool := false;
   END_VAR
   VAR_TEMP   // added for the SCL form of the ladder/FBD networks
      _w1 : Bool;
   END_VAR
BEGIN

REGION Network 1: INIT TEMP
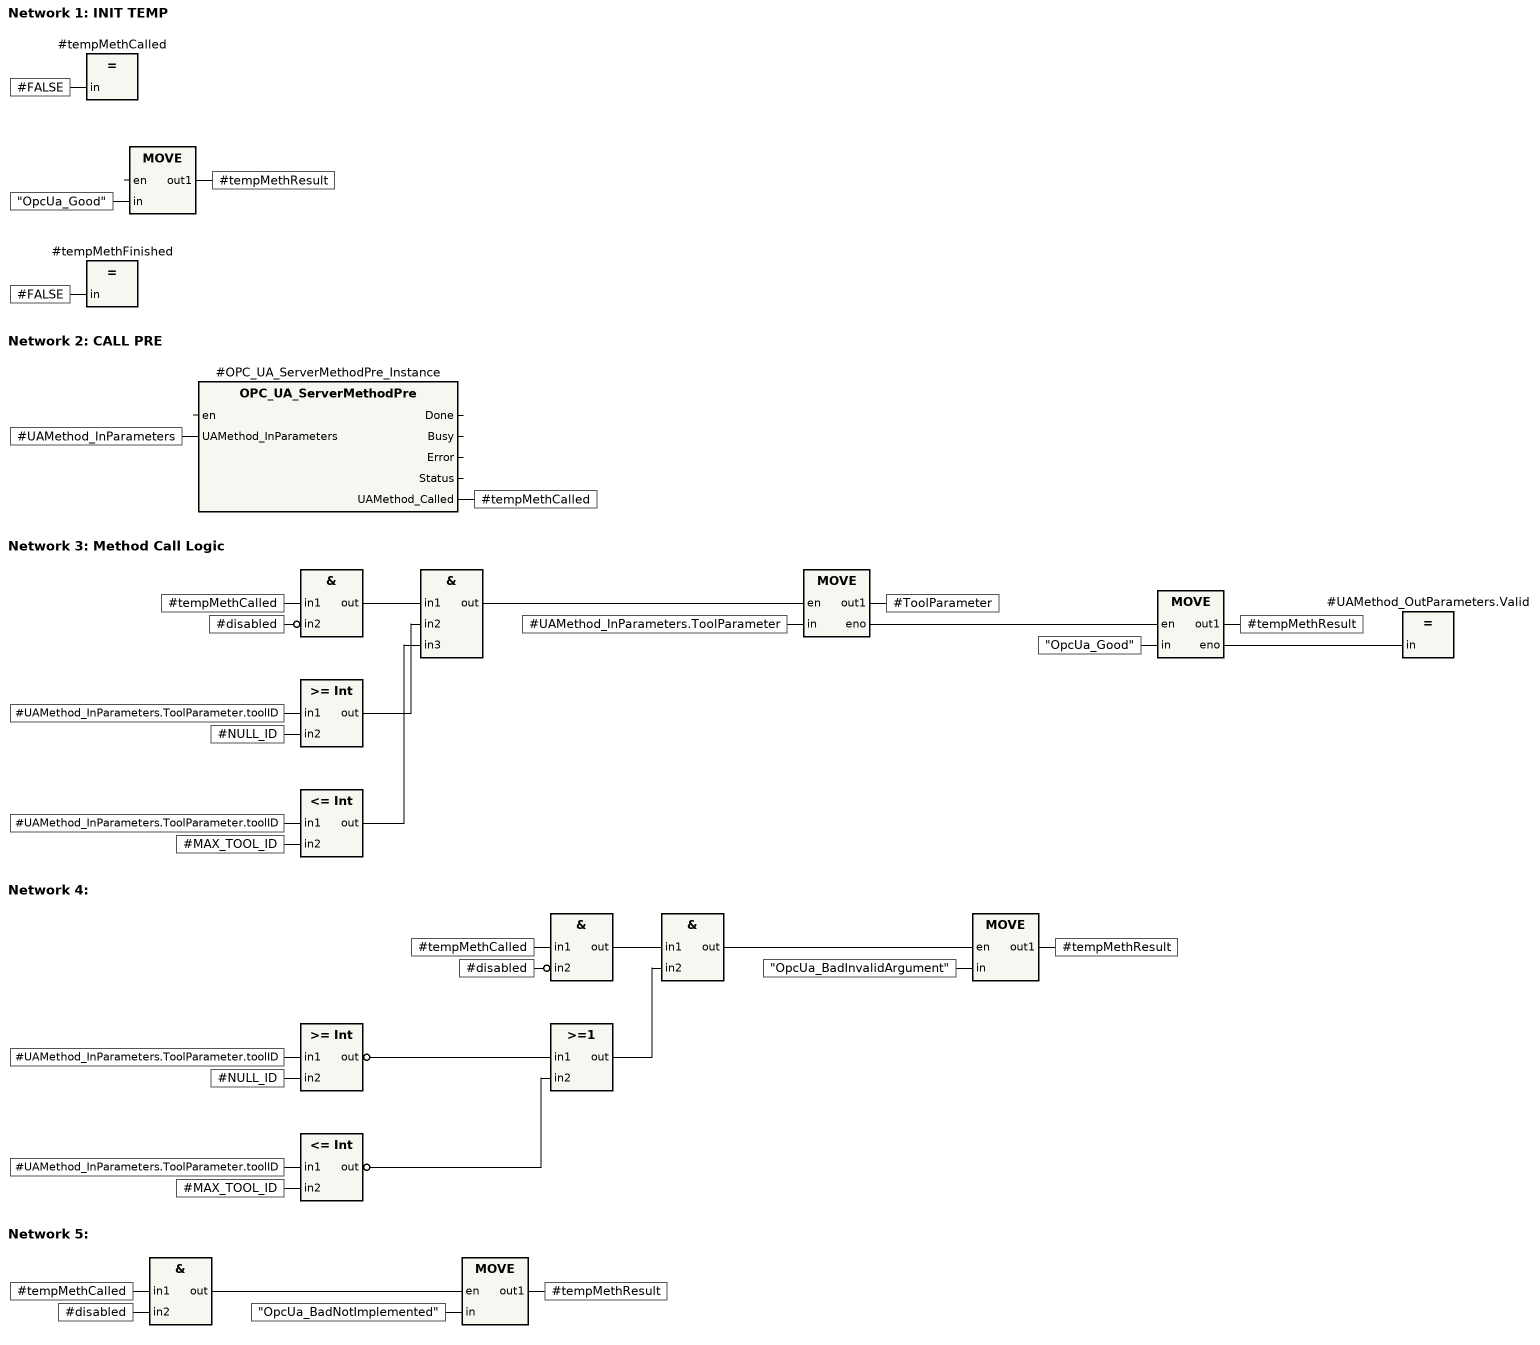
   #tempMethCalled := #FALSE;
   #tempMethResult := "OpcUa_Good";
   #tempMethFinished := #FALSE;
END_REGION

REGION Network 2: CALL PRE
   #OPC_UA_ServerMethodPre_Instance(UAMethod_InParameters := #UAMethod_InParameters,   // OPC_UA_ServerMethodPre
                           UAMethod_Called => #tempMethCalled);
END_REGION

REGION Network 3: Method Call Logic
   // Check input req and if valid set output
   #_w1 := #tempMethCalled AND NOT #disabled AND (#UAMethod_InParameters.ToolParameter.toolID >= #NULL_ID) AND (#UAMethod_InParameters.ToolParameter.toolID <= #MAX_TOOL_ID);
   IF #_w1 THEN
       #ToolParameter := #UAMethod_InParameters.ToolParameter;
       #tempMethResult := "OpcUa_Good";
   END_IF;
   #UAMethod_OutParameters.Valid := #_w1;
END_REGION

REGION Network 4
   // Check input req and if invalid set output
   IF #tempMethCalled AND NOT #disabled AND (NOT (#UAMethod_InParameters.ToolParameter.toolID >= #NULL_ID) OR NOT (#UAMethod_InParameters.ToolParameter.toolID <= #MAX_TOOL_ID)) THEN
       #tempMethResult := "OpcUa_BadInvalidArgument";
   END_IF;
END_REGION

REGION Network 5
   IF #tempMethCalled AND #disabled THEN #tempMethResult := "OpcUa_BadNotImplemented"; END_IF;
END_REGION

REGION Network 6: Set finished to true
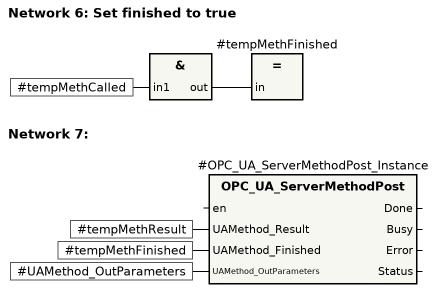
   #tempMethFinished := #tempMethCalled;
END_REGION

REGION Network 7
   #OPC_UA_ServerMethodPost_Instance(UAMethod_Result := #tempMethResult,   // OPC_UA_ServerMethodPost
                           UAMethod_Finished := #tempMethFinished,
                           UAMethod_OutParameters := #UAMethod_OutParameters);
END_REGION
END_FUNCTION_BLOCK

ORGANIZATION_BLOCK "MethodOB"   // OB123, FBD, ProgramCycle
TITLE = "Main Program Sweep (Cycle)"
{ S7_Optimized_Access := 'TRUE' }
VERSION : 0.1
   VAR_INPUT
      Initial_Call : Bool;   // Initial call of this OB
      Remanence : Bool;   // =True, if remanent data are available
   END_VAR
BEGIN

REGION Network 1
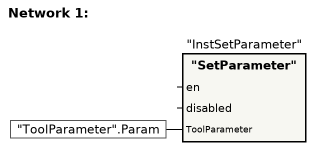
   "InstSetParameter"(ToolParameter := "ToolParameter".Param);   // "SetParameter"
END_REGION
END_ORGANIZATION_BLOCK

// ===== PLC "ZOPCClient@SUP"  CPU 1518-4 PN/DP =====

VAR_GLOBAL   // PLC tag table "StandardVariablentabelle"
   "ClockByte" AT %MB0 : Byte;
   "Clock10Hz" AT %M0.0 : Bool;
   "Clock5Hz" AT %M0.1 : Bool;
   "Clock2.5Hz" AT %M0.2 : Bool;
   "Clock2Hz" AT %M0.3 : Bool;
   "Clock1.25Hz" AT %M0.4 : Bool;
   "Clock1Hz" AT %M0.5 : Bool;
   "Clock0.625Hz" AT %M0.6 : Bool;
   "Clock0.5Hz" AT %M0.7 : Bool;
   "SystemByte" AT %MB1 : Byte;
   "FirstScan" AT %M1.0 : Bool;
   "DiagStatusUpdate" AT %M1.1 : Bool;
   "AlwaysTRUE" AT %M1.2 : Bool;
   "AlwaysFALSE" AT %M1.3 : Bool;
   "ConnectDemo" AT %M10.1 : Bool;
   "ReadDemo" AT %M10.2 : Bool;
   "WriteDemo" AT %M10.3 : Bool;
   "CallMethodDemo" AT %M10.4 : Bool;
   "ConnectClient" AT %M20.0 : Bool;
   "GetNameSpaceIndex" AT %M20.1 : Bool;
   "GetNodeHandle1" AT %M20.2 : Bool;
   "GetNodeHandle2" AT %M20.3 : Bool;
   "GetMethodHandle" AT %M20.4 : Bool;
   "WriteData" AT %M20.5 : Bool;
   "ReadData" AT %M20.6 : Bool;
   "CallMethod" AT %M20.7 : Bool;
   "DisconnectClient" AT %M21.0 : Bool;
END_VAR

VAR_GLOBAL   // PLC tag table "AnalogTags"
   "AI0" AT %EW4 : Word;
   "AI1" AT %EW9 : Word;
   "AI2" AT %EW11 : Word;
   "AI3" AT %EW13 : Word;
   "AI4" AT %EW15 : Word;
   "AI5" AT %EW14 : Word;
   "AI6" AT %EW16 : Word;
   "AI7" AT %EW18 : Word;
   "AO0" AT %AW4 : Word;
   "AO1" AT %AW6 : Word;
   "AO2" AT %AW8 : Word;
   "AO3" AT %AW10 : Word;
END_VAR

VAR_GLOBAL   // PLC tag table "CounterTags"
   "Z1" AT %Z1 : Counter;
   "Z2" AT %Z2 : Counter;
   "Z3" AT %Z3 : Counter;
   "Z4" AT %Z4 : Counter;
   "Z5" AT %Z5 : Counter;
   "Z7" AT %Z7 : Counter;
   "Z8" AT %Z8 : Counter;
   "Z9" AT %Z9 : Counter;
   "Z10" AT %Z10 : Counter;
   "ZTest" AT %Z100 : Counter;
   "Z6" AT %Z6 : Counter;
   "Z500" AT %Z500 : Counter;
   "Z1000" AT %Z1000 : Counter;
   "Z1023" AT %Z1023 : Counter;
   "Z1024" AT %Z1024 : Counter;
   "Z2047" AT %Z2047 : Counter;
END_VAR

VAR_GLOBAL   // PLC tag table "DigitalInputTags"
   "DI01" AT %E0.1 : Bool;
   "DI02" AT %E0.2 : Bool;
   "DI03" AT %E0.3 : Bool;
   "DI04" AT %E0.4 : Bool;
   "DI05" AT %E0.5 : Bool;
   "DI06" AT %E0.6 : Bool;
   "DI07" AT %E0.7 : Bool;
   "DI11" AT %E1.1 : Bool;
   "DI12" AT %E1.2 : Bool;
   "DI13" AT %E1.3 : Bool;
   "DI14" AT %E1.4 : Bool;
   "DI15" AT %E1.5 : Bool;
   "DI16" AT %E1.6 : Bool;
   "DI17" AT %E1.7 : Bool;
   "DI20" AT %E2.0 : Bool;
   "DI21" AT %E2.1 : Bool;
   "DI22" AT %E2.2 : Bool;
   "DI23" AT %E2.3 : Bool;
   "DI24" AT %E2.4 : Bool;
   "DI25" AT %E2.5 : Bool;
   "DI26" AT %E2.6 : Bool;
   "DI27" AT %E2.7 : Bool;
   "DI30" AT %E3.0 : Bool;
   "DI31" AT %E3.1 : Bool;
   "DI32" AT %E3.2 : Bool;
   "DI33" AT %E3.3 : Bool;
   "DI34" AT %E3.4 : Bool;
   "DI35" AT %E3.5 : Bool;
   "DI36" AT %E3.6 : Bool;
   "DI37" AT %E3.7 : Bool;
   "DI10" AT %E1.0 : Bool;
   "DI00" AT %E0.0 : Bool;
   "DI1" AT %EB1 : Byte;
   "DI300" AT %EB300 : Byte;
   "DI310W" AT %EW310 : Word;
   "DI320D" AT %ED320 : DWord;
   "DI3300" AT %E330.0 : Bool;
   "DI340L" AT %E340.0 : LWord;
   "DI0" AT %EB0 : Byte;
END_VAR

VAR_GLOBAL   // PLC tag table "DigitalOutputTags"
   "DO01" AT %A0.1 : Bool;
   "DO02" AT %A0.2 : Bool;
   "DO04" AT %A0.4 : Bool;
   "DO05" AT %A0.5 : Bool;
   "DO06" AT %A0.6 : Bool;
   "DO07" AT %A0.7 : Bool;
   "DO10" AT %A1.0 : Bool;
   "DO11" AT %A1.1 : Bool;
   "DO12" AT %A1.2 : Bool;
   "DO13" AT %A1.3 : Bool;
   "DO14" AT %A1.4 : Bool;
   "DO15" AT %A1.5 : Bool;
   "DO16" AT %A1.6 : Bool;
   "DO17" AT %A1.7 : Bool;
   "DO20" AT %A2.0 : Bool;
   "DO21" AT %A2.1 : Bool;
   "DO22" AT %A2.2 : Bool;
   "DO23" AT %A2.3 : Bool;
   "DO24" AT %A2.4 : Bool;
   "DO25" AT %A2.5 : Bool;
   "DO26" AT %A2.6 : Bool;
   "DO27" AT %A2.7 : Bool;
   "DO30" AT %A3.0 : Bool;
   "DO31" AT %A3.1 : Bool;
   "DO32" AT %A3.2 : Bool;
   "DO33" AT %A3.3 : Bool;
   "DO34" AT %A3.4 : Bool;
   "DO35" AT %A3.5 : Bool;
   "DO36" AT %A3.6 : Bool;
   "DO37" AT %A3.7 : Bool;
   "DO300" AT %AB300 : Byte;
   "DO00" AT %A0.0 : Bool;
   "DO03" AT %A0.3 : Bool;
   "DO120" AT %A12.0 : Bool;
   "DO1" AT %AB1 : Byte;
   "DO0" AT %AB0 : Byte;
   "DOW0" AT %AW0 : Word;
   "DOW2" AT %AW2 : Word;
   "DO310W" AT %AW310 : Word;
   "DO320D" AT %AD320 : DWord;
   "DO3300" AT %A330.0 : Bool;
   "DO340L" AT %A340.0 : LWord;
END_VAR

VAR_GLOBAL   // PLC tag table "MerkerTags"
   "M1000" AT %M100.0 : Bool;
   "M1001" AT %M100.1 : Bool;
   "M1002" AT %M100.2 : Bool;
   "M1003" AT %M100.3 : Bool;
   "M1004" AT %M100.4 : Bool;
   "M1005" AT %M100.5 : Bool;
   "M1006" AT %M100.6 : Bool;
   "M1007" AT %M100.7 : Bool;
   "MB110" AT %MB110 : Byte;
   "MW120" AT %MW120 : Word;
   "MD130" AT %MD130 : DWord;
   "CharMb" AT %MB200 : Char;
   "DateMw" AT %MW202 : Date;
   "DintMd" AT %MD204 : DInt;
   "IntMw" AT %MW208 : Int;
   "LdtMl" AT %M210.0 : LDT;
   "LintMl" AT %M218.0 : LInt;
   "LrealMl" AT %M226.0 : LReal;
   "LtimeMl" AT %M234.0 : LTime;
   "LtodMl" AT %M242.0 : LTime_Of_Day;
   "LwordMl" AT %M250.0 : LWord;
   "RealMd" AT %MD258 : Real;
   "S5timeMw" AT %MW262 : S5Time;
   "SintMb" AT %MB264 : SInt;
   "TimeMd" AT %MD266 : Time;
   "TodMd" AT %MD270 : Time_Of_Day;
   "UdintMd" AT %MD274 : UDInt;
   "UintMw" AT %MW278 : UInt;
   "UlintMl" AT %M280.0 : ULInt;
   "UsintMb" AT %MB288 : USInt;
   "Z1MB" AT %MB500 : Byte;
   "Z2MB" AT %MB501 : Byte;
   "ZTestMx" AT %M502.0 : Bool;
   "Z6FP" AT %M502.1 : Bool;
   "Z7FP" AT %M502.2 : Bool;
   "Z8FP" AT %M502.3 : Bool;
   "Z9FP" AT %M502.4 : Bool;
   "Z10FP" AT %M502.5 : Bool;
   "TremMx" AT %M105.0 : Bool;
   "IintMw400" AT %MW400 : Int;
END_VAR

VAR_GLOBAL   // PLC tag table "TimerTags"
   "T1" AT %T1 : Timer;
   "T3" AT %T3 : Timer;
   "T4" AT %T4 : Timer;
   "T5" AT %T5 : Timer;
   "T6" AT %T6 : Timer;
   "T7" AT %T7 : Timer;
   "T9" AT %T9 : Timer;
   "T10" AT %T10 : Timer;
   "T2" AT %T2 : Timer;
   "T8" AT %T8 : Timer;
   "T20" AT %T20 : Timer;
   "T40" AT %T40 : Timer;
   "T60" AT %T60 : Timer;
   "T80" AT %T80 : Timer;
   "T100" AT %T100 : Timer;
   "T200" AT %T200 : Timer;
   "T500" AT %T500 : Timer;
   "T1000" AT %T1000 : Timer;
   "T2000" AT %T2000 : Timer;
   "T99" AT %T99 : Timer;
   "T85" AT %T85 : Timer;
   "T86" AT %T86 : Timer;
   "T2047" AT %T2047 : Timer;
END_VAR

VAR_GLOBAL CONSTANT   // PLC tag table "Tag table from XML_1"
   "OpcUa_Good" : DWord := 16#00000000;   // Everything is as expected.
   "OpcUa_Uncertain" : DWord := 16#40000000;   // Something unexpected occurred but the results still maybe useable.
   "OpcUa_Bad" : DWord := 16#80000000;   // An error occurred.
   "OpcUa_BadUnexpectedError" : DWord := 16#80010000;   // An unexpected error occurred.
   "OpcUa_BadInternalError" : DWord := 16#80020000;   // An internal error occurred as a result of a programming or configuration error.
   "OpcUa_BadOutOfMemory" : DWord := 16#80030000;   // Not enough memory to complete the operation.
   "OpcUa_BadResourceUnavailable" : DWord := 16#80040000;   // An operating system resource is not available.
   "OpcUa_BadCommunicationError" : DWord := 16#80050000;   // A low level communication error occurred.
   "OpcUa_BadEncodingError" : DWord := 16#80060000;   // Encoding halted because of invalid data in the objects being serialized.
   "OpcUa_BadDecodingError" : DWord := 16#80070000;   // Decoding halted because of invalid data in the stream.
   "OpcUa_BadEncodingLimitsExceeded" : DWord := 16#80080000;   // The message encoding/decoding limits imposed by the stack have been exceeded.
   "OpcUa_BadRequestTooLarge" : DWord := 16#80B80000;   // The request message size exceeds limits set by the server.
   "OpcUa_BadResponseTooLarge" : DWord := 16#80B90000;   // The response message size exceeds limits set by the client.
   "OpcUa_BadUnknownResponse" : DWord := 16#80090000;   // An unrecognized response was received from the server.
   "OpcUa_BadTimeout" : DWord := 16#800A0000;   // The operation timed out.
   "OpcUa_BadServiceUnsupported" : DWord := 16#800B0000;   // The server does not support the requested service.
   "OpcUa_BadShutdown" : DWord := 16#800C0000;   // The operation was cancelled because the application is shutting down.
   "OpcUa_BadServerNotConnected" : DWord := 16#800D0000;   // The operation could not complete because the client is not connected to the server.
   "OpcUa_BadServerHalted" : DWord := 16#800E0000;   // The server has stopped and cannot process any requests.
   "OpcUa_BadNothingToDo" : DWord := 16#800F0000;   // There was nothing to do because the client passed a list of operations with no elements.
   "OpcUa_BadTooManyOperations" : DWord := 16#80100000;   // The request could not be processed because it specified too many operations.
   "OpcUa_BadTooManyMonitoredItems" : DWord := 16#80DB0000;   // The request could not be processed because there are too many monitored items in the subscription.
   "OpcUa_BadDataTypeIdUnknown" : DWord := 16#80110000;   // The extension object cannot be (de)serialized because the data type id is not recognized.
   "OpcUa_BadCertificateInvalid" : DWord := 16#80120000;   // The certificate provided as a parameter is not valid.
   "OpcUa_BadSecurityChecksFailed" : DWord := 16#80130000;   // An error occurred verifying security.
   "OpcUa_BadCertificateTimeInvalid" : DWord := 16#80140000;   // The certificate has expired or is not yet valid.
   "OpcUa_BadCertificateIssuerTimeInvalid" : DWord := 16#80150000;   // An issuer certificate has expired or is not yet valid.
   "OpcUa_BadCertificateHostNameInvalid" : DWord := 16#80160000;   // The HostName used to connect to a server does not match a HostName in the certificate.
   "OpcUa_BadCertificateUriInvalid" : DWord := 16#80170000;   // The URI specified in the ApplicationDescription does not match the URI in the certificate.
   "OpcUa_BadCertificateUseNotAllowed" : DWord := 16#80180000;   // The certificate may not be used for the requested operation.
   "OpcUa_BadCertificateIssuerUseNotAllowed" : DWord := 16#80190000;   // The issuer certificate may not be used for the requested operation.
   "OpcUa_BadCertificateUntrusted" : DWord := 16#801A0000;   // The certificate is not trusted.
   "OpcUa_BadCertificateRevocationUnknown" : DWord := 16#801B0000;   // It was not possible to determine if the certificate has been revoked.
   "OpcUa_BadCertificateIssuerRevocationUnknown" : DWord := 16#801C0000;   // It was not possible to determine if the issuer certificate has been revoked.
   "OpcUa_BadCertificateRevoked" : DWord := 16#801D0000;   // The certificate has been revoked.
   "OpcUa_BadCertificateIssuerRevoked" : DWord := 16#801E0000;   // The issuer certificate has been revoked.
   "OpcUa_BadCertificateChainIncomplete" : DWord := 16#810D0000;   // The certificate chain is incomplete.
   "OpcUa_BadUserAccessDenied" : DWord := 16#801F0000;   // User does not have permission to perform the requested operation.
   "OpcUa_BadIdentityTokenInvalid" : DWord := 16#80200000;   // The user identity token is not valid.
   "OpcUa_BadIdentityTokenRejected" : DWord := 16#80210000;   // The user identity token is valid but the server has rejected it.
   "OpcUa_BadSecureChannelIdInvalid" : DWord := 16#80220000;   // The specified secure channel is no longer valid.
   "OpcUa_BadInvalidTimestamp" : DWord := 16#80230000;   // The timestamp is outside the range allowed by the server.
   "OpcUa_BadNonceInvalid" : DWord := 16#80240000;   // The nonce does appear to be not a random value or it is not the correct length.
   "OpcUa_BadSessionIdInvalid" : DWord := 16#80250000;   // The session id is not valid.
   "OpcUa_BadSessionClosed" : DWord := 16#80260000;   // The session was closed by the client.
   "OpcUa_BadSessionNotActivated" : DWord := 16#80270000;   // The session cannot be used because ActivateSession has not been called.
   "OpcUa_BadSubscriptionIdInvalid" : DWord := 16#80280000;   // The subscription id is not valid.
   "OpcUa_BadRequestHeaderInvalid" : DWord := 16#802A0000;   // The header for the request is missing or invalid.
   "OpcUa_BadTimestampsToReturnInvalid" : DWord := 16#802B0000;   // The timestamps to return parameter is invalid.
   "OpcUa_BadRequestCancelledByClient" : DWord := 16#802C0000;   // The request was cancelled by the client.
   "OpcUa_BadTooManyArguments" : DWord := 16#80E50000;   // Too many arguments were provided.
   "OpcUa_BadLicenseExpired" : DWord := 16#810E0000;   // The server requires a license to operate in general or to perform a service or operation, but existing license is expired.
   "OpcUa_BadLicenseLimitsExceeded" : DWord := 16#810F0000;   // The server has limits on number of allowed operations / objects, based on installed licenses, and these limits where exceeded.
   "OpcUa_BadLicenseNotAvailable" : DWord := 16#81100000;   // The server does not have a license which is required to operate in general or to perform a service or operation.
   "OpcUa_GoodSubscriptionTransferred" : DWord := 16#002D0000;   // The subscription was transferred to another session.
   "OpcUa_GoodCompletesAsynchronously" : DWord := 16#002E0000;   // The processing will complete asynchronously.
   "OpcUa_GoodOverload" : DWord := 16#002F0000;   // Sampling has slowed down due to resource limitations.
   "OpcUa_GoodClamped" : DWord := 16#00300000;   // The value written was accepted but was clamped.
   "OpcUa_BadNoCommunication" : DWord := 16#80310000;   // Communication with the data source is defined, but not established, and there is no last known value available.
   "OpcUa_BadWaitingForInitialData" : DWord := 16#80320000;   // Waiting for the server to obtain values from the underlying data source.
   "OpcUa_BadNodeIdInvalid" : DWord := 16#80330000;   // The syntax of the node id is not valid.
   "OpcUa_BadNodeIdUnknown" : DWord := 16#80340000;   // The node id refers to a node that does not exist in the server address space.
   "OpcUa_BadAttributeIdInvalid" : DWord := 16#80350000;   // The attribute is not supported for the specified Node.
   "OpcUa_BadIndexRangeInvalid" : DWord := 16#80360000;   // The syntax of the index range parameter is invalid.
   "OpcUa_BadIndexRangeNoData" : DWord := 16#80370000;   // No data exists within the range of indexes specified.
   "OpcUa_BadDataEncodingInvalid" : DWord := 16#80380000;   // The data encoding is invalid.
   "OpcUa_BadDataEncodingUnsupported" : DWord := 16#80390000;   // The server does not support the requested data encoding for the node.
   "OpcUa_BadNotReadable" : DWord := 16#803A0000;   // The access level does not allow reading or subscribing to the Node.
   "OpcUa_BadNotWritable" : DWord := 16#803B0000;   // The access level does not allow writing to the Node.
   "OpcUa_BadOutOfRange" : DWord := 16#803C0000;   // The value was out of range.
   "OpcUa_BadNotSupported" : DWord := 16#803D0000;   // The requested operation is not supported.
   "OpcUa_BadNotFound" : DWord := 16#803E0000;   // A requested item was not found or a search operation ended without success.
   "OpcUa_BadObjectDeleted" : DWord := 16#803F0000;   // The object cannot be used because it has been deleted.
   "OpcUa_BadNotImplemented" : DWord := 16#80400000;   // Requested operation is not implemented.
   "OpcUa_BadMonitoringModeInvalid" : DWord := 16#80410000;   // The monitoring mode is invalid.
   "OpcUa_BadMonitoredItemIdInvalid" : DWord := 16#80420000;   // The monitoring item id does not refer to a valid monitored item.
   "OpcUa_BadMonitoredItemFilterInvalid" : DWord := 16#80430000;   // The monitored item filter parameter is not valid.
   "OpcUa_BadMonitoredItemFilterUnsupported" : DWord := 16#80440000;   // The server does not support the requested monitored item filter.
   "OpcUa_BadFilterNotAllowed" : DWord := 16#80450000;   // A monitoring filter cannot be used in combination with the attribute specified.
   "OpcUa_BadStructureMissing" : DWord := 16#80460000;   // A mandatory structured parameter was missing or null.
   "OpcUa_BadEventFilterInvalid" : DWord := 16#80470000;   // The event filter is not valid.
   "OpcUa_BadContentFilterInvalid" : DWord := 16#80480000;   // The content filter is not valid.
   "OpcUa_BadFilterOperatorInvalid" : DWord := 16#80C10000;   // An unregognized operator was provided in a filter.
   "OpcUa_BadFilterOperatorUnsupported" : DWord := 16#80C20000;   // A valid operator was provided, but the server does not provide support for this filter operator.
   "OpcUa_BadFilterOperandCountMismatch" : DWord := 16#80C30000;   // The number of operands provided for the filter operator was less then expected for the operand provided.
   "OpcUa_BadFilterOperandInvalid" : DWord := 16#80490000;   // The operand used in a content filter is not valid.
   "OpcUa_BadFilterElementInvalid" : DWord := 16#80C40000;   // The referenced element is not a valid element in the content filter.
   "OpcUa_BadFilterLiteralInvalid" : DWord := 16#80C50000;   // The referenced literal is not a valid value.
   "OpcUa_BadContinuationPointInvalid" : DWord := 16#804A0000;   // The continuation point provide is longer valid.
   "OpcUa_BadNoContinuationPoints" : DWord := 16#804B0000;   // The operation could not be processed because all continuation points have been allocated.
   "OpcUa_BadReferenceTypeIdInvalid" : DWord := 16#804C0000;   // The operation could not be processed because all continuation points have been allocated.
   "OpcUa_BadBrowseDirectionInvalid" : DWord := 16#804D0000;   // The browse direction is not valid.
   "OpcUa_BadNodeNotInView" : DWord := 16#804E0000;   // The node is not part of the view.
   "OpcUa_BadNumericOverflow" : DWord := 16#81120000;   // The number was not accepted because of a numeric overflow.
   "OpcUa_BadServerUriInvalid" : DWord := 16#804F0000;   // The ServerUri is not a valid URI.
   "OpcUa_BadServerNameMissing" : DWord := 16#80500000;   // No ServerName was specified.
   "OpcUa_BadDiscoveryUrlMissing" : DWord := 16#80510000;   // No DiscoveryUrl was specified.
   "OpcUa_BadSempahoreFileMissing" : DWord := 16#80520000;   // The semaphore file specified by the client is not valid.
   "OpcUa_BadRequestTypeInvalid" : DWord := 16#80530000;   // The security token request type is not valid.
   "OpcUa_BadSecurityModeRejected" : DWord := 16#80540000;   // The security mode does not meet the requirements set by the server.
   "OpcUa_BadSecurityPolicyRejected" : DWord := 16#80550000;   // The security policy does not meet the requirements set by the server.
   "OpcUa_BadTooManySessions" : DWord := 16#80560000;   // The server has reached its maximum number of sessions.
   "OpcUa_BadUserSignatureInvalid" : DWord := 16#80570000;   // The user token signature is missing or invalid.
   "OpcUa_BadApplicationSignatureInvalid" : DWord := 16#80580000;   // The signature generated with the client certificate is missing or invalid.
   "OpcUa_BadNoValidCertificates" : DWord := 16#80590000;   // The client did not provide at least one software certificate that is valid and meets the profile requirements for the server.
   "OpcUa_BadIdentityChangeNotSupported" : DWord := 16#80C60000;   // The server does not support changing the user identity assigned to the session.
   "OpcUa_BadRequestCancelledByRequest" : DWord := 16#805A0000;   // The request was cancelled by the client with the Cancel service.
   "OpcUa_BadParentNodeIdInvalid" : DWord := 16#805B0000;   // The parent node id does not to refer to a valid node.
   "OpcUa_BadReferenceNotAllowed" : DWord := 16#805C0000;   // The reference could not be created because it violates constraints imposed by the data model.
   "OpcUa_BadNodeIdRejected" : DWord := 16#805D0000;   // The requested node id was reject because it was either invalid or server does not allow node ids to be specified by the client.
   "OpcUa_BadNodeIdExists" : DWord := 16#805E0000;   // The requested node id is already used by another node.
   "OpcUa_BadNodeClassInvalid" : DWord := 16#805F0000;   // The node class is not valid.
   "OpcUa_BadBrowseNameInvalid" : DWord := 16#80600000;   // The browse name is invalid.
   "OpcUa_BadBrowseNameDuplicated" : DWord := 16#80610000;   // The browse name is not unique among nodes that share the same relationship with the parent.
   "OpcUa_BadNodeAttributesInvalid" : DWord := 16#80620000;   // The node attributes are not valid for the node class.
   "OpcUa_BadTypeDefinitionInvalid" : DWord := 16#80630000;   // The type definition node id does not reference an appropriate type node.
   "OpcUa_BadSourceNodeIdInvalid" : DWord := 16#80640000;   // The source node id does not reference a valid node.
   "OpcUa_BadTargetNodeIdInvalid" : DWord := 16#80650000;   // The target node id does not reference a valid node.
   "OpcUa_BadDuplicateReferenceNotAllowed" : DWord := 16#80660000;   // The reference type between the nodes is already defined.
   "OpcUa_BadInvalidSelfReference" : DWord := 16#80670000;   // The server does not allow this type of self reference on this node.
   "OpcUa_BadReferenceLocalOnly" : DWord := 16#80680000;   // The reference type is not valid for a reference to a remote server.
   "OpcUa_BadNoDeleteRights" : DWord := 16#80690000;   // The server will not allow the node to be deleted.
   "OpcUa_UncertainReferenceNotDeleted" : DWord := 16#40BC0000;   // The server was not able to delete all target references.
   "OpcUa_BadServerIndexInvalid" : DWord := 16#806A0000;   // The server index is not valid.
   "OpcUa_BadViewIdUnknown" : DWord := 16#806B0000;   // The view id does not refer to a valid view node.
   "OpcUa_BadViewTimestampInvalid" : DWord := 16#80C90000;   // The view timestamp is not available or not supported.
   "OpcUa_BadViewParameterMismatch" : DWord := 16#80CA0000;   // The view parameters are not consistent with each other.
   "OpcUa_BadViewVersionInvalid" : DWord := 16#80CB0000;   // The view version is not available or not supported.
   "OpcUa_UncertainNotAllNodesAvailable" : DWord := 16#40C00000;   // The list of references may not be complete because the underlying system is not available.
   "OpcUa_GoodResultsMayBeIncomplete" : DWord := 16#00BA0000;   // The server should have followed a reference to a node in a remote server but did not. The result set may be incomplete.
   "OpcUa_BadNotTypeDefinition" : DWord := 16#80C80000;   // The provided Nodeid was not a type definition nodeid.
   "OpcUa_UncertainReferenceOutOfServer" : DWord := 16#406C0000;   // One of the references to follow in the relative path references to a node in the address space in another server.
   "OpcUa_BadTooManyMatches" : DWord := 16#806D0000;   // The requested operation has too many matches to return.
   "OpcUa_BadQueryTooComplex" : DWord := 16#806E0000;   // The requested operation requires too many resources in the server.
   "OpcUa_BadNoMatch" : DWord := 16#806F0000;   // The requested operation has no match to return.
   "OpcUa_BadMaxAgeInvalid" : DWord := 16#80700000;   // The max age parameter is invalid.
   "OpcUa_BadSecurityModeInsufficient" : DWord := 16#80E60000;   // The operation is not permitted over the current secure channel.
   "OpcUa_BadHistoryOperationInvalid" : DWord := 16#80710000;   // The history details parameter is not valid.
   "OpcUa_BadHistoryOperationUnsupported" : DWord := 16#80720000;   // The server does not support the requested operation.
   "OpcUa_BadInvalidTimestampArgument" : DWord := 16#80BD0000;   // The defined timestamp to return was invalid.
   "OpcUa_BadWriteNotSupported" : DWord := 16#80730000;   // The server does not support writing the combination of value, status and timestamps provided.
   "OpcUa_BadTypeMismatch" : DWord := 16#80740000;   // The value supplied for the attribute is not of the same type as the attributes value.
   "OpcUa_BadMethodInvalid" : DWord := 16#80750000;   // The method id does not refer to a method for the specified object.
   "OpcUa_BadArgumentsMissing" : DWord := 16#80760000;   // The client did not specify all of the input arguments for the method.
   "OpcUa_BadNotExecutable" : DWord := 16#81110000;   // The executable attribute does not allow the execution of the method.
   "OpcUa_BadTooManySubscriptions" : DWord := 16#80770000;   // The server has reached its maximum number of subscriptions.
   "OpcUa_BadTooManyPublishRequests" : DWord := 16#80780000;   // The server has reached the maximum number of queued publish requests.
   "OpcUa_BadNoSubscription" : DWord := 16#80790000;   // There is no subscription available for this session.
   "OpcUa_BadSequenceNumberUnknown" : DWord := 16#807A0000;   // The sequence number is unknown to the server.
   "OpcUa_BadMessageNotAvailable" : DWord := 16#807B0000;   // The requested notification message is no longer available.
   "OpcUa_BadInsufficientClientProfile" : DWord := 16#807C0000;   // The client of the current session does not support one or more Profiles that are necessary for the subscription.
   "OpcUa_BadStateNotActive" : DWord := 16#80BF0000;   // The sub-state machine is not currently active.
   "OpcUa_BadTcpServerTooBusy" : DWord := 16#807D0000;   // The server cannot process the request because it is too busy.
   "OpcUa_BadTcpMessageTypeInvalid" : DWord := 16#807E0000;   // The type of the message specified in the header invalid.
   "OpcUa_BadTcpSecureChannelUnknown" : DWord := 16#807F0000;   // The SecureChannelId and/or TokenId are not currently in use.
   "OpcUa_BadTcpMessageTooLarge" : DWord := 16#80800000;   // The size of the message specified in the header is too large.
   "OpcUa_BadTcpNotEnoughResources" : DWord := 16#80810000;   // There are not enough resources to process the request.
   "OpcUa_BadTcpInternalError" : DWord := 16#80820000;   // An internal error occurred.
   "OpcUa_BadTcpEndpointUrlInvalid" : DWord := 16#80830000;   // The server does not recognize the QueryString specified.
   "OpcUa_BadRequestInterrupted" : DWord := 16#80840000;   // The request could not be sent because of a network interruption.
   "OpcUa_BadRequestTimeout" : DWord := 16#80850000;   // Timeout occurred while processing the request.
   "OpcUa_BadSecureChannelClosed" : DWord := 16#80860000;   // The secure channel has been closed.
   "OpcUa_BadSecureChannelTokenUnknown" : DWord := 16#80870000;   // The token has expired or is not recognized.
   "OpcUa_BadSequenceNumberInvalid" : DWord := 16#80880000;   // The sequence number is not valid.
   "OpcUa_BadProtocolVersionUnsupported" : DWord := 16#80BE0000;   // The applications do not have compatible protocol versions.
   "OpcUa_BadConfigurationError" : DWord := 16#80890000;   // There is a problem with the configuration that affects the usefulness of the value.
   "OpcUa_BadNotConnected" : DWord := 16#808A0000;   // The variable should receive its value from another variable, but has never been configured to do so.
   "OpcUa_BadDeviceFailure" : DWord := 16#808B0000;   // There has been a failure in the device/data source that generates the value that has affected the value.
   "OpcUa_BadSensorFailure" : DWord := 16#808C0000;   // There has been a failure in the sensor from which the value is derived by the device/data source.
   "OpcUa_BadOutOfService" : DWord := 16#808D0000;   // The source of the data is not operational.
   "OpcUa_BadDeadbandFilterInvalid" : DWord := 16#808E0000;   // The deadband filter is not valid.
   "OpcUa_UncertainNoCommunicationLastUsableValue" : DWord := 16#408F0000;   // Communication to the data source has failed. The variable value is the last value that had a good quality.
   "OpcUa_UncertainLastUsableValue" : DWord := 16#40900000;   // Whatever was updating this value has stopped doing so.
   "OpcUa_UncertainSubstituteValue" : DWord := 16#40910000;   // The value is an operational value that was manually overwritten.
   "OpcUa_UncertainInitialValue" : DWord := 16#40920000;   // The value is an initial value for a variable that normally receives its value from another variable.
   "OpcUa_UncertainSensorNotAccurate" : DWord := 16#40930000;   // The value is at one of the sensor limits.
   "OpcUa_UncertainEngineeringUnitsExceeded" : DWord := 16#40940000;   // The value is outside of the range of values defined for this parameter.
   "OpcUa_UncertainSubNormal" : DWord := 16#40950000;   // The value is derived from multiple sources and has less than the required number of Good sources.
   "OpcUa_GoodLocalOverride" : DWord := 16#00960000;   // The value has been overridden.
   "OpcUa_BadRefreshInProgress" : DWord := 16#80970000;   // This Condition refresh failed, a Condition refresh operation is already in progress.
   "OpcUa_BadConditionAlreadyDisabled" : DWord := 16#80980000;   // This condition has already been disabled.
   "OpcUa_BadConditionAlreadyEnabled" : DWord := 16#80CC0000;   // This condition has already been enabled.
   "OpcUa_BadConditionDisabled" : DWord := 16#80990000;   // Property not available, this condition is disabled.
   "OpcUa_BadEventIdUnknown" : DWord := 16#809A0000;   // The specified event id is not recognized.
   "OpcUa_BadEventNotAcknowledgeable" : DWord := 16#80BB0000;   // The event cannot be acknowledged.
   "OpcUa_BadDialogNotActive" : DWord := 16#80CD0000;   // The dialog condition is not active.
   "OpcUa_BadDialogResponseInvalid" : DWord := 16#80CE0000;   // The response is not valid for the dialog.
   "OpcUa_BadConditionBranchAlreadyAcked" : DWord := 16#80CF0000;   // The condition branch has already been acknowledged.
   "OpcUa_BadConditionBranchAlreadyConfirmed" : DWord := 16#80D00000;   // The condition branch has already been confirmed.
   "OpcUa_BadConditionAlreadyShelved" : DWord := 16#80D10000;   // The condition has already been shelved.
   "OpcUa_BadConditionNotShelved" : DWord := 16#80D20000;   // The condition is not currently shelved.
   "OpcUa_BadShelvingTimeOutOfRange" : DWord := 16#80D30000;   // The shelving time not within an acceptable range.
   "OpcUa_BadNoData" : DWord := 16#809B0000;   // No data exists for the requested time range or event filter.
   "OpcUa_BadBoundNotFound" : DWord := 16#80D70000;   // No data found to provide upper or lower bound value.
   "OpcUa_BadBoundNotSupported" : DWord := 16#80D80000;   // The server cannot retrieve a bound for the variable.
   "OpcUa_BadDataLost" : DWord := 16#809D0000;   // Data is missing due to collection started/stopped/lost.
   "OpcUa_BadDataUnavailable" : DWord := 16#809E0000;   // Expected data is unavailable for the requested time range due to an un-mounted volume, an off-line archive or tape, or similar reason for temporary unavailability.
   "OpcUa_BadEntryExists" : DWord := 16#809F0000;   // The data or event was not successfully inserted because a matching entry exists.
   "OpcUa_BadNoEntryExists" : DWord := 16#80A00000;   // The data or event was not successfully updated because no matching entry exists.
   "OpcUa_BadTimestampNotSupported" : DWord := 16#80A10000;   // The client requested history using a timestamp format the server does not support (i.e requested ServerTimestamp when server only supports SourceTimestamp).
   "OpcUa_GoodEntryInserted" : DWord := 16#00A20000;   // The data or event was successfully inserted into the historical database.
   "OpcUa_GoodEntryReplaced" : DWord := 16#00A30000;   // The data or event field was successfully replaced in the historical database.
   "OpcUa_UncertainDataSubNormal" : DWord := 16#40A40000;   // The value is derived from multiple values and has less than the required number of Good values.
   "OpcUa_GoodNoData" : DWord := 16#00A50000;   // No data exists for the requested time range or event filter.
   "OpcUa_GoodMoreData" : DWord := 16#00A60000;   // The data or event field was successfully replaced in the historical database.
   "OpcUa_BadAggregateListMismatch" : DWord := 16#80D40000;   // The requested number of Aggregates does not match the requested number of NodeIds.
   "OpcUa_BadAggregateNotSupported" : DWord := 16#80D50000;   // The requested Aggregate is not support by the server.
   "OpcUa_BadAggregateInvalidInputs" : DWord := 16#80D60000;   // The aggregate value could not be derived due to invalid data inputs.
   "OpcUa_BadAggregateConfigurationRejected" : DWord := 16#80DA0000;   // The aggregate configuration is not valid for specified node.
   "OpcUa_GoodDataIgnored" : DWord := 16#00D90000;   // The request pecifies fields which are not valid for the EventType or cannot be saved by the historian.
   "OpcUa_BadRequestNotAllowed" : DWord := 16#80E40000;   // The request was rejected by the server because it did not meet the criteria set by the server.
   "OpcUa_BadRequestNotComplete" : DWord := 16#81130000;   // The request has not been processed by the server yet.
   "OpcUa_GoodEdited" : DWord := 16#00DC0000;   // The value does not come from the real source and has been edited by the server.
   "OpcUa_GoodPostActionFailed" : DWord := 16#00DD0000;   // There was an error in execution of these post-actions.
   "OpcUa_UncertainDominantValueChanged" : DWord := 16#40DE0000;   // The related EngineeringUnit has been changed but the Variable Value is still provided based on the previous unit.
   "OpcUa_GoodDependentValueChanged" : DWord := 16#00E00000;   // A dependent value has been changed but the change has not been applied to the device.
   "OpcUa_BadDominantValueChanged" : DWord := 16#80E10000;   // The related EngineeringUnit has been changed but this change has not been applied to the device. The Variable Value is still dependent on the previous unit but its status is currently Bad.
   "OpcUa_UncertainDependentValueChanged" : DWord := 16#40E20000;   // A dependent value has been changed but the change has not been applied to the device. The quality of the dominant variable is uncertain.
   "OpcUa_BadDependentValueChanged" : DWord := 16#80E30000;   // A dependent value has been changed but the change has not been applied to the device. The quality of the dominant variable is Bad.
   "OpcUa_GoodCommunicationEvent" : DWord := 16#00A70000;   // The communication layer has raised an event.
   "OpcUa_GoodShutdownEvent" : DWord := 16#00A80000;   // The system is shutting down.
   "OpcUa_GoodCallAgain" : DWord := 16#00A90000;   // The operation is not finished and needs to be called again.
   "OpcUa_GoodNonCriticalTimeout" : DWord := 16#00AA0000;   // A non-critical timeout occurred.
   "OpcUa_BadInvalidArgument" : DWord := 16#80AB0000;   // One or more arguments are invalid.
   "OpcUa_BadConnectionRejected" : DWord := 16#80AC0000;   // Could not establish a network connection to remote server.
   "OpcUa_BadDisconnect" : DWord := 16#80AD0000;   // The server has disconnected from the client.
   "OpcUa_BadConnectionClosed" : DWord := 16#80AE0000;   // The network connection has been closed.
   "OpcUa_BadInvalidState" : DWord := 16#80AF0000;   // The operation cannot be completed because the object is closed, uninitialized or in some other invalid state.
   "OpcUa_BadEndOfStream" : DWord := 16#80B00000;   // Cannot move beyond end of the stream.
   "OpcUa_BadNoDataAvailable" : DWord := 16#80B10000;   // No data is currently available for reading from a non-blocking stream.
   "OpcUa_BadWaitingForResponse" : DWord := 16#80B20000;   // The asynchronous operation is waiting for a response.
   "OpcUa_BadOperationAbandoned" : DWord := 16#80B30000;   // The asynchronous operation was abandoned by the caller.
   "OpcUa_BadExpectedStreamToBlock" : DWord := 16#80B40000;   // The stream did not return all data requested (possibly because it is a non-blocking stream).
   "OpcUa_BadWouldBlock" : DWord := 16#80B50000;   // Non blocking behaviour is required and the operation would block.
   "OpcUa_BadSyntaxError" : DWord := 16#80B60000;   // A value had an invalid syntax.
   "OpcUa_BadMaxConnectionsReached" : DWord := 16#80B70000;   // The operation could not be finished because all available connections are in use.
END_VAR

TYPE "typeToolParameter"
   STRUCT
      length : Int;
      width : Int;
      weight : Int;
      toolID : Int;
   END_STRUCT;
END_TYPE

// folder: SystemDataTypeFolder

TYPE "Client interface_1.Read Machine Data"
   STRUCT
      Speed : LReal;
      Parts : DInt;
      Frequency : Real;
      length : Int;
      width : Int;
      weight : Int;
      toolID : Int;
   END_STRUCT;
END_TYPE

TYPE "Client interface_1.Control Machine"
   STRUCT
      Run : Bool;
   END_STRUCT;
END_TYPE

TYPE "Client interface_1.Set Machine Tool Parameter.Method.Inputs"
   STRUCT
      ToolParameter : "typeToolParameter";
   END_STRUCT;
END_TYPE

TYPE "Client interface_1.Set Machine Tool Parameter.Method.Outputs"
   STRUCT
      Valid : Bool;
   END_STRUCT;
END_TYPE

// folder: 10_Demo_OpcClient

DATA_BLOCK "InstOpcUaClient"   // DB1
{ S7_Optimized_Access := 'TRUE' }
AUTHOR : SiemensAG
VERSION : 1.0
// stored: InstanceOfName OpcUaClient
"OpcUaClient"
BEGIN
END_DATA_BLOCK

DATA_BLOCK "Client interface_1_Data"   // DB3
{ S7_Optimized_Access := 'TRUE' }
VERSION : 0.1
   VAR
      "Read Machine Data" : Struct
         Variable : "Client interface_1.Read Machine Data";
         NodeStatusList : Array[0..6] of DWord;
         TimeStamps : Array[0..6] of LDT;
      END_STRUCT;
      "Control Machine" : Struct
         Variable : "Client interface_1.Control Machine";
         NodeStatusList : Array[0..0] of DWord;
      END_STRUCT;
      "Set Machine Tool Parameter" : Struct
         MethodStatusList : Array[0..0] of DWord;
         MethodResultList : Array[0..0] of DWord;
         Method : Struct
            Inputs : "Client interface_1.Set Machine Tool Parameter.Method.Inputs";
            Outputs : "Client interface_1.Set Machine Tool Parameter.Method.Outputs";
         END_STRUCT;
      END_STRUCT;
   END_VAR
BEGIN
END_DATA_BLOCK

// folder: System blocks/Program resources

DATA_BLOCK "Client interface_1_Configuration"   // DB2
{ S7_Optimized_Access := 'TRUE' }
VERSION : 0.1
   VAR
      Connection : Struct
         ConnectInfo : OPC_UA_SessionConnectInfo;
         ConnectionHdl : DWord;
         ServerEndpointUrl : String[254] := 'opc.tcp://10.11.28.70:4840';
      END_STRUCT;
      Namespaces : Struct
         NamespaceURIs : Array[0..0] of WString;
         ServerNamespaceIndexes : Array[0..0] of UInt;
         NamespaceStatusList : Array[0..0] of DWord;
         NamespaceCount : UInt := 1;
      END_STRUCT;
      ReadLists : Struct
         "Read Machine Data" : Struct
            NodeCount : UInt := 7;
            Nodes : Array[0..6] of OPC_UA_NodeId;
            NodeHdls : Array[0..6] of DWord;
         END_STRUCT;
      END_STRUCT;
      WriteLists : Struct
         "Control Machine" : Struct
            NodeCount : UInt := 1;
            Nodes : Array[0..0] of OPC_UA_NodeId;
            NodeHdls : Array[0..0] of DWord;
         END_STRUCT;
      END_STRUCT;
      MethodLists : Struct
         "Set Machine Tool Parameter" : Struct
            MethodCount : UInt := 1;
            ObjectNodes : Array[0..0] of OPC_UA_NodeId;
            MethodNodes : Array[0..0] of OPC_UA_NodeId;
            MethodHdls : Array[0..0] of DWord;
         END_STRUCT;
      END_STRUCT;
   END_VAR
BEGIN
   ReadLists."Read Machine Data".Nodes[0].NamespaceIndex := 0;
   ReadLists."Read Machine Data".Nodes[0].IdentifierType := 1;
   ReadLists."Read Machine Data".Nodes[0].Identifier := WSTRING#'"MachineParameter"."Speed"';
   ReadLists."Read Machine Data".Nodes[1].NamespaceIndex := 0;
   ReadLists."Read Machine Data".Nodes[1].IdentifierType := 1;
   ReadLists."Read Machine Data".Nodes[1].Identifier := WSTRING#'"MachineParameter"."Parts"';
   ReadLists."Read Machine Data".Nodes[2].NamespaceIndex := 0;
   ReadLists."Read Machine Data".Nodes[2].IdentifierType := 1;
   ReadLists."Read Machine Data".Nodes[2].Identifier := WSTRING#'"MachineParameter"."Frequency"';
   ReadLists."Read Machine Data".Nodes[3].NamespaceIndex := 0;
   ReadLists."Read Machine Data".Nodes[3].IdentifierType := 1;
   ReadLists."Read Machine Data".Nodes[3].Identifier := WSTRING#'"ToolParameter"."Param"."length"';
   ReadLists."Read Machine Data".Nodes[4].NamespaceIndex := 0;
   ReadLists."Read Machine Data".Nodes[4].IdentifierType := 1;
   ReadLists."Read Machine Data".Nodes[4].Identifier := WSTRING#'"ToolParameter"."Param"."width"';
   ReadLists."Read Machine Data".Nodes[5].NamespaceIndex := 0;
   ReadLists."Read Machine Data".Nodes[5].IdentifierType := 1;
   ReadLists."Read Machine Data".Nodes[5].Identifier := WSTRING#'"ToolParameter"."Param"."weight"';
   ReadLists."Read Machine Data".Nodes[6].NamespaceIndex := 0;
   ReadLists."Read Machine Data".Nodes[6].IdentifierType := 1;
   ReadLists."Read Machine Data".Nodes[6].Identifier := WSTRING#'"ToolParameter"."Param"."toolID"';
   WriteLists."Control Machine".Nodes[0].NamespaceIndex := 0;
   WriteLists."Control Machine".Nodes[0].IdentifierType := 1;
   WriteLists."Control Machine".Nodes[0].Identifier := WSTRING#'"MachineControl"."Run"';
   MethodLists."Set Machine Tool Parameter".MethodNodes[0].NamespaceIndex := 0;
   MethodLists."Set Machine Tool Parameter".MethodNodes[0].IdentifierType := 1;
   MethodLists."Set Machine Tool Parameter".MethodNodes[0].Identifier := WSTRING#'"InstSetParameter".Method';
   MethodLists."Set Machine Tool Parameter".ObjectNodes[0].NamespaceIndex := 0;
   MethodLists."Set Machine Tool Parameter".ObjectNodes[0].IdentifierType := 1;
   MethodLists."Set Machine Tool Parameter".ObjectNodes[0].Identifier := WSTRING#'"InstSetParameter"';
   Connection.ConnectInfo.SessionName := WSTRING#'OPC UA Connection_1';
   Connection.ConnectInfo.ApplicationName := WSTRING#'';
   Connection.ConnectInfo.SecurityMsgMode := 1;
   Connection.ConnectInfo.SecurityPolicy := 1;
   Connection.ConnectInfo.ServerUri := '';
   Connection.ConnectInfo.CheckServerCertificate := False;
   Connection.ConnectInfo.TransportProfile := 1;
   Connection.ConnectInfo.UserIdentityTokenType := 0;
   Connection.ConnectInfo.CertificateID := 0;
   Connection.ConnectInfo.SessionTimeout := T#30S;
   Connection.ConnectInfo.MonitorConnection := T#5S;
   Connection.ConnectInfo.LocaleIDs[0] := 'de-DE';
   Connection.ConnectInfo.LocaleIDs[1] := '';
   Connection.ConnectInfo.LocaleIDs[2] := '';
   Connection.ConnectInfo.LocaleIDs[3] := '';
   Connection.ConnectInfo.LocaleIDs[4] := '';
   Namespaces.NamespaceURIs[0] := WSTRING#'http://www.siemens.com/simatic-s7-opcua';
END_DATA_BLOCK

// folder: (top level)

ORGANIZATION_BLOCK "Main"   // OB1, FBD, ProgramCycle
TITLE = "Main Program Sweep (Cycle)"
{ S7_Optimized_Access := 'TRUE' }
VERSION : 0.1
   VAR_INPUT
      Initial_Call : Bool;   // Initial call of this OB
      Remanence : Bool;   // =True, if remanent data are available
   END_VAR
BEGIN

REGION Network 1: OPC UA Connect
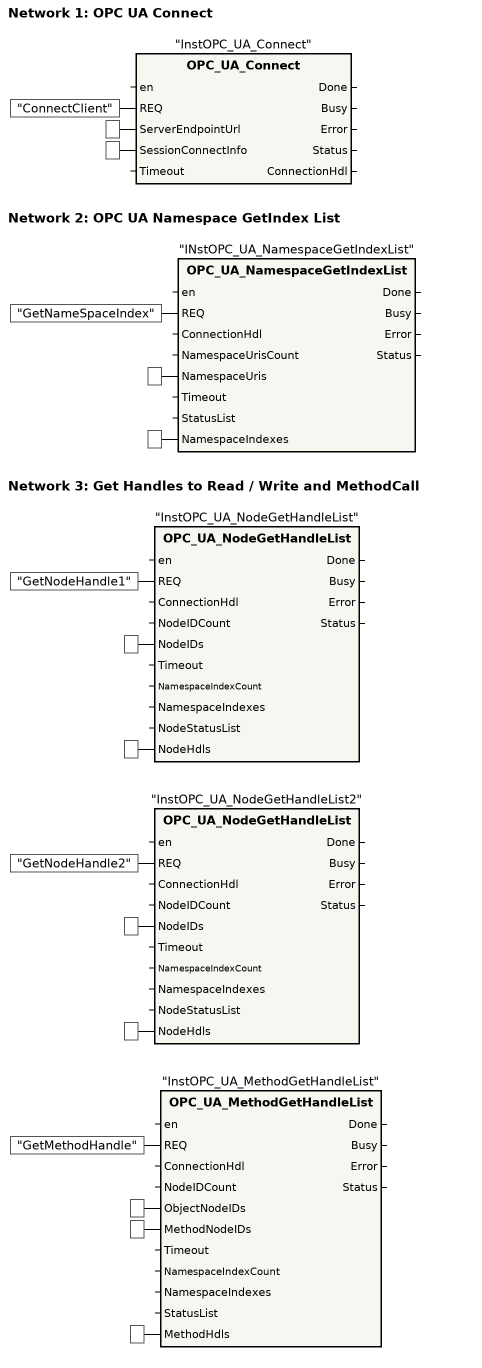
   // no checked SCL form for this network; see the picture
END_REGION

REGION Network 2: OPC UA Namespace GetIndex List
   // no checked SCL form for this network; see the picture
END_REGION

REGION Network 3: Get Handles to Read / Write and MethodCall
   // no checked SCL form for this network; see the picture
END_REGION

REGION Network 4: Write Data with OPC UA Client
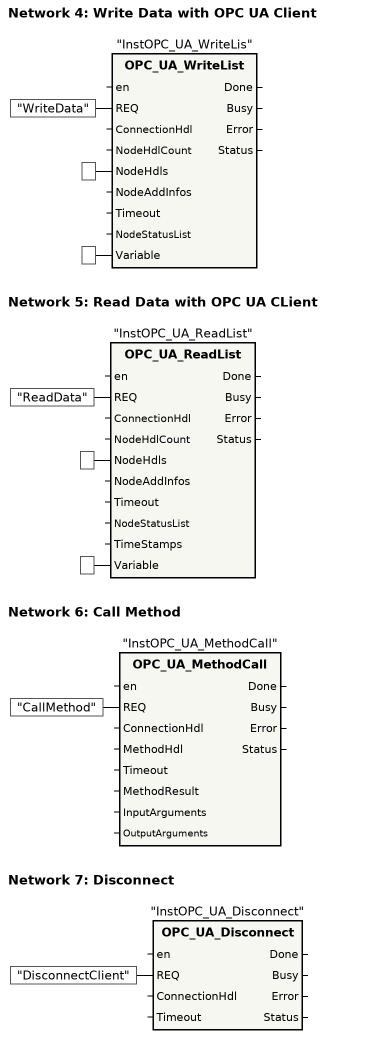
   // no checked SCL form for this network; see the picture
END_REGION

REGION Network 5: Read Data with OPC UA CLient
   // no checked SCL form for this network; see the picture
END_REGION

REGION Network 6: Call Method
   "InstOPC_UA_MethodCall"(REQ := "CallMethod");   // OPC_UA_MethodCall
END_REGION

REGION Network 7: Disconnect
   "InstOPC_UA_Disconnect"(REQ := "DisconnectClient");   // OPC_UA_Disconnect
END_REGION

REGION Network 8: OpcUaClient
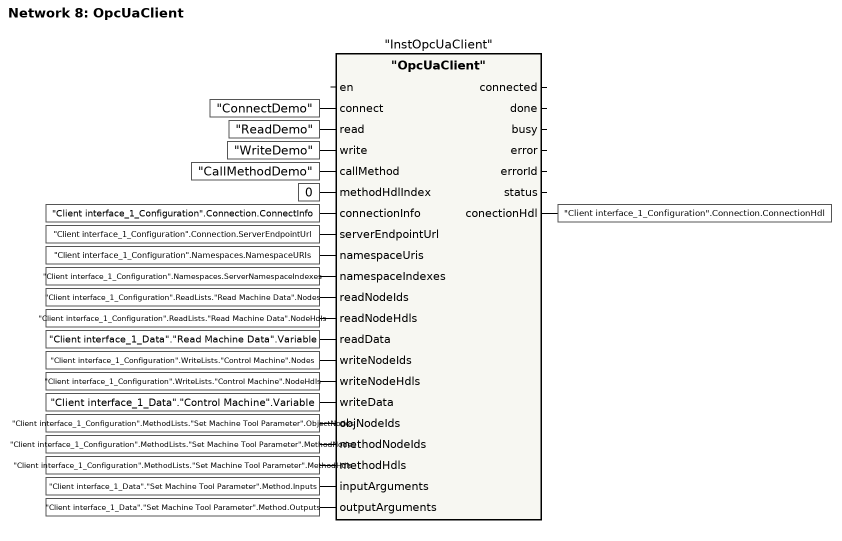
   "InstOpcUaClient"(connect := "ConnectDemo",   // "OpcUaClient"
                     read := "ReadDemo",
                     write := "WriteDemo",
                     callMethod := "CallMethodDemo",
                     methodHdlIndex := 0,
                     connectionInfo := "Client interface_1_Configuration".Connection.ConnectInfo,
                     serverEndpointUrl := "Client interface_1_Configuration".Connection.ServerEndpointUrl,
                     namespaceUris := "Client interface_1_Configuration".Namespaces.NamespaceURIs,
                     namespaceIndexes := "Client interface_1_Configuration".Namespaces.ServerNamespaceIndexes,
                     readNodeIds := "Client interface_1_Configuration".ReadLists."Read Machine Data".Nodes,
                     readNodeHdls := "Client interface_1_Configuration".ReadLists."Read Machine Data".NodeHdls,
                     readData := "Client interface_1_Data"."Read Machine Data".Variable,
                     writeNodeIds := "Client interface_1_Configuration".WriteLists."Control Machine".Nodes,
                     writeNodeHdls := "Client interface_1_Configuration".WriteLists."Control Machine".NodeHdls,
                     writeData := "Client interface_1_Data"."Control Machine".Variable,
                     objNodeIds := "Client interface_1_Configuration".MethodLists."Set Machine Tool Parameter".ObjectNodes,
                     methodNodeIds := "Client interface_1_Configuration".MethodLists."Set Machine Tool Parameter".MethodNodes,
                     methodHdls := "Client interface_1_Configuration".MethodLists."Set Machine Tool Parameter".MethodHdls,
                     inputArguments := "Client interface_1_Data"."Set Machine Tool Parameter".Method.Inputs,
                     outputArguments := "Client interface_1_Data"."Set Machine Tool Parameter".Method.Outputs,
                     conectionHdl => "Client interface_1_Configuration".Connection.ConnectionHdl);
END_REGION
END_ORGANIZATION_BLOCK

// folder: 10_Demo_OpcClient

FUNCTION_BLOCK "OpcUaClient"   // FB2, SCL
TITLE = OpcUaClient
{ S7_Optimized_Access := 'TRUE' }
AUTHOR : SiemensAG
VERSION : 1.0
// OPC UA-Client-Wrapper
   VAR_INPUT
      connect : Bool;
      read : Bool;
      write : Bool;
      callMethod : Bool;
      methodHdlIndex : DInt;
      connectionInfo : OPC_UA_SessionConnectInfo;
      serverEndpointUrl : String;
   END_VAR
   VAR_OUTPUT
      connected : Bool;
      done : Bool;
      busy : Bool;
      error : Bool;
      errorId : Int;
      status : DWord;
      conectionHdl : DWord;
   END_VAR
   VAR_IN_OUT
      namespaceUris : Variant;
      namespaceIndexes : Variant;
      readNodeIds : Variant;
      readNodeHdls : Variant;
      readData : Variant;
      writeNodeIds : Variant;
      writeNodeHdls : Variant;
      writeData : Variant;
      objNodeIds : Variant;
      methodNodeIds : Variant;
      methodHdls : Variant;
      inputArguments : Variant;
      outputArguments : Variant;
   END_VAR
   VAR
      instOpcUaConnect : OPC_UA_Connect;
      instOpcUaConnectionGetStatus : OPC_UA_ConnectionGetStatus;
      instOpcUaNamespaceGIL : OPC_UA_NamespaceGetIndexList;
      InstOpcUaGHLRead : OPC_UA_NodeGetHandleList;
      instOpcUaGHLWrite : OPC_UA_NodeGetHandleList;
      instOpcUaGHLMethods : OPC_UA_MethodGetHandleList;
      InstOpcUaRHLRead : OPC_UA_NodeReleaseHandleList;
      instOpcUaRHLWrite : OPC_UA_NodeReleaseHandleList;
      instOpcUaRHLMethods : OPC_UA_MethodReleaseHandleList;
      instOpcUaReadList : OPC_UA_ReadList;
      instOpcUaWriteList : OPC_UA_WriteList;
      instOpcUaMethodCall : OPC_UA_MethodCall;
      instOpcUaDisconnect : OPC_UA_Disconnect;
      instConnRTrig : R_TRIG;
      instDisconRTrig : R_TRIG;
      instReconTrigger : R_TRIG;
      instNGILTrigger : R_TRIG;
      instReadTrigger : R_TRIG;
      instWriteTrigger : R_TRIG;
      instMethodCallTrigger : R_TRIG;
      instClearConnTrig : R_TRIG;
      statCase : Int;
      statDone : Bool;
      statConnected : Bool;
      statBusy : Bool;
      statError : Bool;
      statErrorId : Int;
      statStatus : DWord;
      statOpcUaRequests : Struct
         Connect : Bool;
         ConGS : Bool;
         NGIL : Bool;
         GHLRead : Bool;
         GHLMethods : Bool;
         GHLWrite : Bool;
         Read : Bool;
         Write : Bool;
         MethodCall : Bool;
         RHLRead : Bool;
         RHLWrite : Bool;
         RHLMethods : Bool;
         Disconnect : Bool;
      END_STRUCT;
      statRHLTrigger : Bool;
      statConnectCount : Int;
      statNamespaceIndexesSet : Bool;
      statNamespaceRegCount : Int;
      statRegisteredRead : Bool;
      statRegisterCountRead : Int;
      statRegisteredWrite : Bool;
      statRegisterCountWrite : Int;
      statRegisteredMethods : Bool;
      statRegisterCountMethod : Int;
      statReadCount : Int;
      statWriteCount : Int;
      statMethodCallCount : DWord;
      statMethodResult : DWord;
      statMethodHdl : DWord;
      statMethodHdlId : DInt;
      statConnectionHdl : DWord;
      instCycDiag : TON_TIME;
      statCycDiagTrigger : Bool;
      statOpcUaReadTimeStamps : Array[0..299] of LDT;
      statSerializeMethodHdls : Array[0..1199] of Byte;
      statOpcUaStatusLists : Struct
         MethodRHL : Array[0..299] of DWord;
         MethodGHL : Array[0..299] of DWord;
         WriteRHL : Array[0..299] of DWord;
         WriteList : Array[0..299] of DWord;
         WriteGHL : Array[0..299] of DWord;
         ReadRHL : Array[0..299] of DWord;
         ReadList : Array[0..299] of DWord;
         ReadGHL : Array[0..299] of DWord;
         NamespaceGIL : Array[0..299] of DWord;
      END_STRUCT;
   END_VAR
   VAR_TEMP
      tempConnectTrigger : Bool;
      tempDisconnectTrigger : Bool;
      tempIndex : Int;
      tempReadTrigger : Bool;
      tempWriteTrigger : Bool;
      tempMethodCallTrigger : Bool;
      tempRetVal : Int;
      tempCycDiag : Bool;
      tempReconnectTrigger : Bool;
      tempRHLTrigger : Bool;
   END_VAR
   VAR CONSTANT
      CASE_CONNECT : Int := 0;
      CASE_NAMESPACE_GET_INDEX_LIST : Int := 1;
      CASE_CONNECTION_GET_STATUS : Int := 2;
      CASE_NODE_GET_HANDLE_LIST : Int := 3;
      CASE_CONNECTED : Int := 4;
      UACS_CONNECTED : UDInt := 0;
      UASS_RUNNING : UDInt := 0;
      UASL_GOOD : UDInt := 16#0000_00FF;
      STATUS_SESSION_CLEANEDUP : DWord := 16#A000_0105;
      STATUS_BUSY : Word := 16#7001;
      STATUS_SERVER_NOT_CONNECTED : DWord := 16#800D_0000;
      STATUS_BAD_CONNECTION_CLOSED : DWord := 16#80AE_0000;
      STATUS_IDLE : Word := 16#7000;
      STATUS_NOT_REGISTERED : Word := 16#80FF;
      STATUS_DONE : Word := 16#0000;
      CYC_TIME_GCS : Time := T#5S;
      OPC_UA_FUNCTIONS_TIMEOUT : Time := T#10S;
      ERR_ID_GOOD : SInt := 0;
      ERR_ID_CON : SInt := 1;
      ERR_ID_CON_GS_STATUS : SInt := 10;
      ERR_ID_CON_GS_CSTATE : SInt := 11;
      ERR_ID_CON_GS_SSTATE : SInt := 12;
      ERR_ID_CON_GS_SLVL : SInt := 13;
      ERR_ID_NGIL : SInt := 2;
      ERR_ID_R_GHL : SInt := 31;
      ERR_ID_W_GHL : SInt := 32;
      ERR_ID_M_GHL : SInt := 33;
      ERR_ID_RL : SInt := 4;
      ERR_ID_WL : SInt := 5;
      ERR_ID_MC : SInt := 6;
      ERR_ID_R_RHL : SInt := 71;
      ERR_ID_W_RHL : SInt := 72;
      ERR_ID_M_RHL : SInt := 73;
      ERR_ID_DISCON : SInt := 8;
   END_VAR
BEGIN
   //=============================================================================
   // Siemens AG (c)Copyright (2019)
   //-----------------------------------------------------------------------------
   // Library: -
   // Tested with: CPU 1513-1 PN;  FW 2.6
   // Engineering: TIA Portal (V15.1)
   // Restrictions: -
   // Requirements: OPC UA Client activated, Fimware V2.6; Set PLC time
   // Functionality: Encapsulates OPC UA client blocks for read, write and method
   //                call including connection handling and diagnosis
   //-----------------------------------------------------------------------------
   // Change log table:
   // Version    Date         Expert in charge           Changes applied
   // 01.00.00   01.02.2019   Siemens SUP Applications   First released version
   //=============================================================================


   //State machine
   CASE #statCase OF
     #CASE_CONNECT:
       REGION Connection Handling
         //initialize FB
         IF NOT #connect THEN
           #statError := FALSE;
           #statBusy := FALSE;
           #statDone := FALSE;
           #statConnected := FALSE;
           #statErrorId := #ERR_ID_GOOD;
           #statStatus := #STATUS_DONE;
         END_IF;

         //Rising Edge detection of connect
         #instConnRTrig(CLK := #connect,
                        Q => #tempConnectTrigger);

         #instReconTrigger(CLK := #connect
                           AND NOT #statConnected
                           AND (#statStatus = #STATUS_SESSION_CLEANEDUP OR #statStatus = #STATUS_BAD_CONNECTION_CLOSED),
                           Q => #tempReconnectTrigger);

